    # the path for welding a floor straight weld with v chisels on both sides.
    # start at the right side and move left.
    def calculate_straight_points_floor(struct1, floorthick, leftpointteach, rightpointteach):
        # get the stuff
        point0 = struct1[0]
        p0x = point0[0]
        p0y = point0[1]
        p0z = point0[2]
        v3xunit = struct1[1]
        v3yunit = struct1[2]
        v3zunit = struct1[3]
        heading1 = struct1[4]
        v4xunit = struct1[5]
        v4yunit = struct1[6]
        lpy = leftpointteach[1]
        rpy = rightpointteach[1]

        # first, check if we need a lift column raise
        # (we do not, because the floors are low)
        zpi = p0z
        floorz = zpi

        # calculate pointtopvcham (left point) (tilted and tiltraised)
        chamferup = floorthick * 25.4 / 1000.0
        tiltraise = 0.006 # 6 mm raise needed for the tip to clear the plane during tiltback
        # on this one, move the tiltraise distance sideways (towards robot) and the chamferover distance up
        x = p0x + v4xunit * tiltraise * -1
        y = p0y + v4yunit * tiltraise * -1
        z = floorz + chamferup

        # calculate rxryrz for tilted back
        # 3 rotations to make this happen.
        # start point is straight up with the preheat pointed in the +y direction.
        # first rotation is 90 degrees about y axis. positive direction. gun is now pointing in the x+ direction with preheat facing +y direction
        m1 = get_rotation_matrix_from_description("y", 1, 90 * pi / 180)
        # second rotation is about 180 degrees about the z axis. heading1 plus 90 degrees. gun is now pointing directly into the sidewall
        m2 = get_rotation_matrix_from_description("z", 1, pi/2 + heading1)
        # third rotation is 10 degrees about the z axis. gun is now tilted back 10 degrees from the sidewall
        m3 = get_rotation_matrix_from_description("z", 1, 10 * pi / 180)
        # combine them by multiplying m3 * m2 * m1
        # matrix multiplication is not commutative but it IS associative, so you can do this whichever order
        m4 = multiply_matrix(m2, m1)
        m5 = multiply_matrix(m3, m4)
        rxryrzt = convert_matrix_to_axang(m5)
        rxt = rxryrzt[0]
        ryt = rxryrzt[1]
        rzt = rxryrzt[2]
        # the non tilted angle is just m4
        rxryrz = convert_matrix_to_axang(m4)
        rx = rxryrz[0]
        ry = rxryrz[1]
        rz = rxryrz[2]
        pointtopvcham = p[x, y, z, rxt, ryt, rzt]

        # calculate distance between leftpoint and rightpoint
        # we have the y distance. we need to find the total distance.
        # the unit vector (v3) should have a magnitude of 1. that's what analyze_touchpoints_only_cover_straight() calculated.
        # so the total distance is y distance * 1 / v3yunit
        ydist = rpy - lpy
        totdist = ydist / v3yunit

        # calculate pointtopvcham2 (right point) (tilted and tiltraised)
        x2 = x + v3xunit * totdist
        y2 = y + v3yunit * totdist
        z2 = z + v3zunit * totdist
        pointtopvcham2 = p[x2, y2, z2, rxt, ryt, rzt]

        # calculate point1 (preheat)
        dist = 1 * 25.4 / 1000.0 # move back 1 inch from ptvc2 (in this case back means positive)
        p1x = x2 + dist * v3xunit
        p1y = y2 + dist * v3yunit
        p1z = z2 + dist * v3zunit
        point1 = p[p1x, p1y, p1z, rxt, ryt, rzt]

        # calculate point2 (start of flatten)
        dist = -0.5 * 25.4 / 1000.0  # half an inch past the top of v chamfer
        p2x = x2 + dist * v3xunit
        p2y = y2 + dist * v3yunit
        p2z = z2 + dist * v3zunit
        point2 = p[p2x, p2y, p2z, rxt, ryt, rzt]

        # calculate point3 (end of flatten)
        dist = -1.5 * 25.4 / 1000.0  # 1.5 inches past top of v chamfer
        p3x = x2 + dist * v3xunit + tiltraise * v4xunit
        p3y = y2 + dist * v3yunit + tiltraise * v4yunit
        p3z = z2 + dist * v3zunit
        point3 = p[p3x, p3y, p3z, rx, ry, rz]

        # calculate point4 (start of unflatten)
        dist = 1.5 * 25.4 / 1000.0
        p4x = x + v3xunit * dist + tiltraise * v4xunit
        p4y = y + v3yunit * dist + tiltraise * v4yunit
        p4z = z + v3zunit * dist
        point4 = p[p4x, p4y, p4z, rx, ry, rz]

        # calculate point5 (end of unflatten)
        dist = 0.5 * 25.4 / 1000.0
        p5x = x + v3xunit * dist
        p5y = y + v3yunit * dist
        p5z = z + v3zunit * dist
        point5 = p[p5x, p5y, p5z, rxt, ryt, rzt]

        # calculate point6 (end of smear)
        dist = -2 * 25.4 / 1000.0
        p6x = x + v3xunit * dist
        p6y = y + v3yunit * dist
        p6z = z + v3zunit * dist
        point6 = p[p6x, p6y, p6z, rxt, ryt, rzt]

        # return struct
        ret = struct(pointtopvcham=pointtopvcham, point1=point1, point2=point2, point3=point3, point4=point4, point5=point5, point6=point6)
        return ret

    end

    # this function determines the starting touchpoints for homing in on cover lt geometry
    # includes two points above the cover lt, closer to the robot than the lt, facing down
    def get_coverlt_homing_pathpoints(leftpoint, rightpoint):
        # get the teach position points
        lpx = leftpoint[0]
        lpy = leftpoint[1]
        lpz = leftpoint[2]
        rpx = rightpoint[0]
        rpy = rightpoint[1]
        rpz = rightpoint[2]

        # specify the distances from (in meters)
        d0 = 0.05 # how far from the cover to approach from
        d1 = 0.03 # how far the touchpints are pushed closer to the robot
        d2 = 0.00 # how far inwards the touchpoints are pushed

        # rxryrz
        rxryrz = [0.334, 3.124, 0]
        rx = rxryrz[0]
        ry = rxryrz[1]
        rz = rxryrz[2]

        # calculate the points
        ph1 = p[lpx + d1, lpy + d2, lpz + d0, rx, ry, rz] # left side approach
        ph2 = p[rpx + d1, rpy - d2, rpz + d0, rx, ry, rz] # right side approach

        ret = struct(ph1=ph1, ph2=ph2)
        is_robot_at_reachable_spot(leftpoint, ret)
        return ret
    end

    def main_calculate_cover_lt(p11, p12, leftpoint, rightpoint):
        struct1 = analyze_touchpoints_only_cover_lt(p11, p12, leftpoint, rightpoint)
        struct2 = calculate_points_cover_lt(struct1)
        #struct2 = calculate_DOtA_points_left_extended(struct1, list1, chamferover, chamferup, tcp_pose_top)
        #struct3 = check_validity_left(struct1, struct2)
        return struct2

    end

    def analyze_touchpoints_only_cover_lt(p11, p12, leftpoint, rightpoint):
        # calculate the slope of the groove in xy plane
        l1p1x = leftpoint[0]
        l1p1y = leftpoint[1]
        l1p2x = rightpoint[0]
        l1p2y = rightpoint[1]

        # equate the first line in 2d space
        ml1 = (l1p2y-l1p1y) / (l1p2x-l1p1x)

        # b = y - mx
        bl1 = l1p1y - ml1 * l1p1x

        # zraise (how much the z value changes from left point to right point
        zraise = p12[2] - p11[2]

        #get the calcpoints
        leftcalcpoint = [leftpoint[0], leftpoint[1], p11[2]]
        rightcalcpoint = [rightpoint[0], rightpoint[1], p12[2]]
        # get the vector from a to b
        vec = [rightcalcpoint[0] - leftcalcpoint[0], rightcalcpoint[1] - leftcalcpoint[1], rightcalcpoint[2] - leftcalcpoint[2]]
        # get the unit vector in 3d
        mag3d = sqrt(vec[0]*vec[0]+vec[1]*vec[1]+vec[2]*vec[2])
        vec3dunit = [vec[0]/mag3d, vec[1]/mag3d, vec[2]/mag3d]
        # get the unit vector in 2d
        mag2d = sqrt(vec[0]*vec[0]+vec[1]*vec[1])
        vec2dunit = [vec[0]/mag2d, vec[1]/mag2d]
        # get the heading
        heading1 = convert_uv_to_heading(vec2dunit[0], vec2dunit[1])

        ret = struct(leftcalcpoint=leftcalcpoint, rightcalcpoint=rightcalcpoint, vxunit=vec3dunit[0], vyunit=vec3dunit[1], vzunit=vec3dunit[2], heading1=heading1)
        return ret
    end

    def calculate_points_cover_lt(struct1):
        # get the stuff from struct
        leftcalcpoint = struct1[0]
        x = leftcalcpoint[0]
        y = leftcalcpoint[1]
        z = leftcalcpoint[2]
        rightcalcpoint = struct1[1]
        x2 = rightcalcpoint[0]
        y2 = rightcalcpoint[1]
        z2 = rightcalcpoint[2]
        v3xunit = struct1[2]
        v3yunit = struct1[3]
        v3zunit = struct1[4]
        heading1 = struct1[5]

        # first calculate rxryrz f normal and tiltback
        # calculate rxryrz for tilted back
        # 3 rotations to make this happen.
        # start point is straight up with the preheat pointed in the +y direction.
        # first rotation is 180 degrees about x direction. gun is now pointing straight down with preheat facing -y direction
        m1 = get_rotation_matrix_from_description("x", 1, 180 * pi / 180)
        # second rotation is a 10 degree turn about the x axis (negative direction)
        m2 = get_rotation_matrix_from_description("x", -1, 10 * pi / 180)
        # third rotation is about 180 degrees about the z axis. starting from the -y axis, go until you get to heading1. that will equal heading1 plus 90 degrees
        m3 = get_rotation_matrix_from_description("z", 1, pi/2 + heading1)
        # combine them by multiplying m3 * m2 * m1
        # matrix multiplication is not commutative but it IS associative, so you can do this whichever order
        m4 = multiply_matrix(m2, m1)
        m5 = multiply_matrix(m3, m4)
        rxryrzt = convert_matrix_to_axang(m5)
        rxt = rxryrzt[0]
        ryt = rxryrzt[1]
        rzt = rxryrzt[2]

        # calculate rxryrz for nontilted
        # first rotation is 180 degrees about x direction. gun is now pointing straight down with preheat facing -y direction
        m1 = get_rotation_matrix_from_description("x", 1, 180 * pi / 180)
        # third rotation is about 180 degrees about the z axis. starting from the -y axis, go until you get to heading1. that will equal heading1 plus 90 degrees
        m3 = get_rotation_matrix_from_description("z", 1, pi/2 + heading1)
        m5 = multiply_matrix(m3, m1)
        rxryrz = convert_matrix_to_axang(m5)
        rx = rxryrz[0]
        ry = rxryrz[1]
        rz = rxryrz[2]

        tiltraise = 0.006 # 6 mm raise needed for the tip to clear the plane during tiltback

        # calculate points 1-3
        # calculate point1 (preheat)
        dist = -1 * 25.4 / 1000.0 # move back 1 inch from
        p1x = x + dist * v3xunit
        p1y = y + dist * v3yunit
        p1z = z + dist * v3zunit + tiltraise
        point1 = p[p1x, p1y, p1z, rxt, ryt, rzt]

        # calculate point2 (start of flatten)
        dist = 0.5 * 25.4 / 1000.0  # half an inch past the top of v chamfer
        p2x = x + dist * v3xunit
        p2y = y + dist * v3yunit
        p2z = z + dist * v3zunit + tiltraise
        point2 = p[p2x, p2y, p2z, rxt, ryt, rzt]

        # calculate point3 (end of flatten)
        dist = 1.5 * 25.4 / 1000.0  # 1.5 inches past top of v chamfer
        p3x = x + dist * v3xunit
        p3y = y + dist * v3yunit
        p3z = z + dist * v3zunit
        point3 = p[p3x, p3y, p3z, rx, ry, rz]

        # calculate points 4-6
        # calculate point4 (start of unflatten)
        dist = -1.5 * 25.4 / 1000.0
        p4x = x2 + v3xunit * dist
        p4y = y2 + v3yunit * dist
        p4z = z2 + v3zunit * dist
        point4 = p[p4x, p4y, p4z, rx, ry, rz]

        # calculate point5 (end of unflatten)
        dist = -0.5 * 25.4 / 1000.0
        p5x = x2 + v3xunit * dist
        p5y = y2 + v3yunit * dist
        p5z = z2 + v3zunit * dist + tiltraise
        point5 = p[p5x, p5y, p5z, rxt, ryt, rzt]

        # calculate point6 (end of smear)
        dist = 2 * 25.4 / 1000.0
        p6x = x2 + v3xunit * dist
        p6y = y2 + v3yunit * dist
        p6z = z2 + v3zunit * dist + tiltraise
        point6 = p[p6x, p6y, p6z, rxt, ryt, rzt]

        # return struct
        ret = struct(pointtopvcham=leftcalcpoint, point1=point1, point2=point2, point3=point3, point4=point4, point5=point5, point6=point6)
        return ret

    end

    def main_calculate_sleeve_fillet(p1, p2, p3):
        struct1 = analyze_touchpoints_only_sleeve_fillet(p1, p2, p3)
        struct2 = calculate_points_sleeve_fillet(struct1)
        return struct2
    end

    # given 3 points at the intersection of the sleeve and the sidewall, this calculates and returns 3 things:
    # the centerpoint of the circle on the plane, the normal vector of the plane, and the radius of the circle
    # then it returns 4 more things after converting to a vertical circle/plane: heading1 (into the plane), vecn, vecr, vecu
    def analyze_touchpoints_only_sleeve_fillet(p1, p2, p3):
        x1 = p1[0]
        y1 = p1[1]
        z1 = p1[2]
        x2 = p2[0]
        y2 = p2[1]
        z2 = p2[2]
        x3 = p3[0]
        y3 = p3[1]
        z3 = p3[2]

        # calculate plane
        # calculate ab (1->2) vector
        abvec = [x2-x1, y2-y1, z2-z1]
        # calculate ac (1->3) vector
        acvec = [x3-x1, y3-y1, z3-z1]
        #calculate the plane's normal vector = ab x ac

        n = crossproduct(abvec, acvec)
        mag = sqrt(n[0]*n[0]+n[1]*n[1]+n[2]*n[2])
        n = [n[0]/mag, n[1]/mag, n[2]/mag]
        d = n[0] * x1 + n[1] * y1 + n[2] * z1

        # find the circle
        # Midpoint of AB:
        mab = [(x1 + x2)/2, (y1 + y2)/2, (z1 + z2)/2]
        # midpoint of ac
        mac = [(x3 + x1)/2, (y3 + y1)/2, (z3 + z1)/2]
        # Get Normal Vectors to AB and AC in the Plane
        # nab (normal to ab) = abvec x n
        nab = crossproduct(abvec, n)
        # nac (normal to ac) = acvec x n
        nac = crossproduct(acvec, n)
        # Define Perpendicular Bisector Lines
        # Each line goes through a midpoint and extends in the direction of the na_
        # we already have the equations of those lines in point vector form with l1 = mab + s * nab, and l2 = mac + t * nac
        # define all the terms so the math is simpler when i have to do math
        mabx = mab[0]
        maby = mab[1]
        mabz = mab[2]
        nabx = nab[0]
        naby = nab[1]
        nabz = nab[2]
        macx = mac[0]
        macy = mac[1]
        macz = mac[2]
        nacx = nac[0]
        nacy = nac[1]
        nacz = nac[2]
        # find the intersection point using the y and z equations
        # maby + s * naby = macy + t * nacy
        # mabz + s * nabz = macz + t * nacz
        # first solve for s and take
        # t = (macz*naby + maby*nabz - mabz*naby - macy*nabz) / (nacy*nabz - naby*nacz)
        t = (macz*naby + maby*nabz - mabz*naby - macy*nabz) / (nacy*nabz - naby*nacz)
        # s = (t*nacz + macz - mabz) / nabz
        s = (t*nacz + macz - mabz) / nabz
        # find the point
        # pcenter = mac + t * nac
        pcenterx = macx + t * nacx
        pcentery = macy + t * nacy
        pcenterz = macz + t * nacz
        rxryrz = [0.528, 4.631, 0.258] # demo point of the welder pointing forward into a sleeve
        pcenter = p[pcenterx, pcentery, pcenterz, rxryrz[0], rxryrz[1], rxryrz[2]]
        radius = distance_between(pcenterx, pcentery, pcenterz, x1, y1, z1)

        # ------ start calculation of vertical assumption -----
        # assume the plane close to vertical
        # fix it to make it actually vertical
        # calculate the unit vector of up, and the unit vector of right.
        # calculate the heading from the +x axis to pointing straight into the wall.
        # the unit vector of up is [0, 0, 1] (because the plane is verticalized) (for easier calculations)
        # first calculate the normal vector INTO the sidewall (make sure x is negative) and make it a unit vector
        vecn = [n[0], n[1], 0] # vector normal
        if vecn[0] > 0:
            vecn = [-n[0], -n[1], 0]
        end
        mag = sqrt(vecn[0]*vecn[0]+vecn[1]*vecn[1])
        vecn = [vecn[0]/mag, vecn[1]/mag, 0]
        # next calculate the right normal vector (the vector IN the plane that goes to the right)
        vecr = [vecn[1], -1*vecn[0], 0]
        vecu = [0, 0, 1] # vector up
        heading1 = convert_uv_to_heading(vecn[0], vecn[1])


        ret = struct(pcenter=pcenter, planenormalvec=n, radius=radius, heading1=heading1, vecn=vecn, vecr=vecr, vecu=vecu)
        return ret
    end

    def crossproduct(vec1, vec2):
        nx = vec1[1]*vec2[2] - vec1[2]*vec2[1]
        ny = vec1[2]*vec2[0] - vec1[0]*vec2[2]
        nz = vec1[0]*vec2[1] - vec1[1]*vec2[0]
        ret = [nx, ny, nz]
        return ret
    end

    # this function calculates only the four points of the quadrants, for the not real program.
    # these calculations are easier so that's why i'm starting with them first.
    # this assumes a vertical plane
    def calculate_points_sleeve_fillet_quadonly(struct1):
        # get the stuff from the struct
        pcenter = struct1[0]
        pcx = pcenter[0]
        pcy = pcenter[1]
        pcz = pcenter[2]
        planenormalvec = struct1[1]
        radius = struct1[2]
        heading1 = struct1[3]
        vecn = struct1[4]
        vecnx = vecn[0]
        vecny = vecn[1]
        vecr = struct1[5]
        vecrx = vecr[0]
        vecry = vecr[1]
        vecu = struct1[6]
        vecuz = vecu[2]

        # define cushions (the backofhole can't actually touch the intersection of pipe and wall, it travels a certain distance around it
        cushout = 0.006 # 5mm # the cushion out from the wall
        cusharound = 0.006 # 5mm # the cushion around the sleeve.

        # get the top point (point1)
        # take the center point and move up the radius plus the cushions
        p1x = pcx + vecnx * -1 * cushout
        p1y = pcy + vecny * -1 * cushout
        p1z = pcz + vecuz * radius + vecuz * cusharound

        # find rxryrz1
        # first rotation is 135 degrees about the y- direction. 90 degrees to get flat. Tip pointing x-, preheat pointing y+. 45 more degrees to get at that above angle
        m1 = get_rotation_matrix_from_description("y", -1, 135 * pi / 180)
        # second rotation is heading1 – 180 degrees about the z+ axis to get pointing straight into wall. Heading1 should be about 180 degrees
        m2 = get_rotation_matrix_from_description("z", 1, heading1 - 180 * pi/180)
        # combine them by multiplying
        m3 = multiply_matrix(m2, m1)
        rxryrz1 = convert_matrix_to_axang(m3)
        rx1 = rxryrz1[0]
        ry1 = rxryrz1[1]
        rz1 = rxryrz1[2]

        point1 = p[p1x, p1y, p1z, rx1, ry1, rz1]

        # get second point (right) (point2)
        # take the center point and move right the radius plus the cushions
        p2x = pcx + vecrx * radius + vecrx * cusharound + vecnx * -1 * cushout
        p2y = pcy + vecry * radius + vecry * cusharound + vecny * -1 * cushout
        p2z = pcz

        # find rxryrz2
        # first rotation is 90 degrees about the x- axis
        m1 = get_rotation_matrix_from_description("x", -1, 90 * pi / 180)
        # second rotation is About 135 degrees about the z+ axis. This calculation is heading1 – 45 degrees
        m2 = get_rotation_matrix_from_description("z", 1, heading1 - 45 * pi/180)
        # combine them by multiplying
        m3 = multiply_matrix(m2, m1)
        rxryrz2 = convert_matrix_to_axang(m3)
        rx2 = rxryrz2[0]
        ry2 = rxryrz2[1]
        rz2 = rxryrz2[2]

        point2 = p[p2x, p2y, p2z, rx2, ry2, rz2]

        # get the third point (bottom) (point3)
        p3x = pcx + vecnx * -1 * cushout
        p3y = pcy + vecny * -1 * cushout
        p3z = pcz - vecuz * radius - vecuz * cusharound

        # find rxryrz3
        # first rotation is 45 degrees about the y+ axis
        m1 = get_rotation_matrix_from_description("y", 1, 45 * pi / 180)
        # second rotation is About 180 degrees about the z+ axis. This calculation is heading1 degrees
        m2 = get_rotation_matrix_from_description("z", 1, heading1)
        # combine them by multiplying
        m3 = multiply_matrix(m2, m1)
        rxryrz3 = convert_matrix_to_axang(m3)
        rx3 = rxryrz3[0]
        ry3 = rxryrz3[1]
        rz3 = rxryrz3[2]

        point3 = p[p3x, p3y, p3z, rx3, ry3, rz3]

        # get the fourth point (left) (point4)
        p4x = pcx - vecrx * radius - vecrx * cusharound + vecnx * -1 * cushout
        p4y = pcy - vecry * radius - vecry * cusharound + vecny * -1 * cushout
        p4z = pcz

        # find rxryrz4
        # first rotation is 90 degrees about the x+ axis
        m1 = get_rotation_matrix_from_description("x", 1, 90 * pi / 180)
        # second rotation is heading1 + 45 degrees about the z+ axis. approx 225 degrees ccw
        m2 = get_rotation_matrix_from_description("z", 1, heading1 + 45 * pi/180)
        # combine them by multiplying
        m3 = multiply_matrix(m2, m1)
        rxryrz4 = convert_matrix_to_axang(m3)
        rx4 = rxryrz4[0]
        ry4 = rxryrz4[1]
        rz4 = rxryrz4[2]

        point4 = p[p4x, p4y, p4z, rx4, ry4, rz4]

        # return the points
        ret = struct(point1=point1, point2=point2, point3=point3, point4=point4)
        return ret

    end

    # this function calculates the points necessary for the fillet sleeve weld path.
    # this assumes a vertical plane
    def calculate_points_sleeve_fillet(struct1):
        # get the stuff from the struct
        pcenter = struct1[0]
        pcx = pcenter[0]
        pcy = pcenter[1]
        pcz = pcenter[2]
        planenormalvec = struct1[1]
        radius = struct1[2]
        heading1 = struct1[3]
        vecn = struct1[4]
        vecnx = vecn[0]
        vecny = vecn[1]
        vecr = struct1[5]
        vecrx = vecr[0]
        vecry = vecr[1]
        vecu = struct1[6]
        vecuz = vecu[2]

        # define cushions (the backofhole can't actually touch the intersection of pipe and wall, it travels a certain distance around it
        cushout = 0.006 # 5mm # the cushion out from the wall
        cusharound = 0.006 # 5mm # the cushion around the sleeve.

        # get the top point (point1)
        # take the center point and move up the radius plus the cushions
        p1x = pcx + vecnx * -1 * cushout
        p1y = pcy + vecny * -1 * cushout
        p1z = pcz + vecuz * radius + vecuz * cusharound

        # find rxryrz1
        # first rotation is 135 degrees about the y- direction. 90 degrees to get flat. Tip pointing x-, preheat pointing y+. 45 more degrees to get at that above angle
        m1 = get_rotation_matrix_from_description("y", -1, 135 * pi / 180)
        # second rotation is heading1 – 180 degrees about the z+ axis to get pointing straight into wall. Heading1 should be about 180 degrees
        m2 = get_rotation_matrix_from_description("z", 1, heading1 - 180 * pi/180)
        # combine them by multiplying
        m3 = multiply_matrix(m2, m1)
        rxryrz1 = convert_matrix_to_axang(m3)
        rx1 = rxryrz1[0]
        ry1 = rxryrz1[1]
        rz1 = rxryrz1[2]

        point1 = p[p1x, p1y, p1z, rx1, ry1, rz1]

        # get second point (right) (point2)
        # take the center point and move right the radius plus the cushions
        p2x = pcx + vecrx * radius + vecrx * cusharound + vecnx * -1 * cushout
        p2y = pcy + vecry * radius + vecry * cusharound + vecny * -1 * cushout
        p2z = pcz

        # find rxryrz2
        # first rotation is 90 degrees about the x- axis
        m1 = get_rotation_matrix_from_description("x", -1, 90 * pi / 180)
        # second rotation is About 135 degrees about the z+ axis. This calculation is heading1 – 45 degrees
        m2 = get_rotation_matrix_from_description("z", 1, heading1 - 45 * pi/180)
        # combine them by multiplying
        m3 = multiply_matrix(m2, m1)
        rxryrz2 = convert_matrix_to_axang(m3)
        rx2 = rxryrz2[0]
        ry2 = rxryrz2[1]
        rz2 = rxryrz2[2]

        point2 = p[p2x, p2y, p2z, rx2, ry2, rz2]

        # get the third point (bottom) (point3)
        p3x = pcx + vecnx * -1 * cushout
        p3y = pcy + vecny * -1 * cushout
        p3z = pcz - vecuz * radius - vecuz * cusharound

        # find rxryrz3
        # first rotation is 45 degrees about the y+ axis
        m1 = get_rotation_matrix_from_description("y", 1, 45 * pi / 180)
        # second rotation is About 180 degrees about the z+ axis. This calculation is heading1 degrees
        m2 = get_rotation_matrix_from_description("z", 1, heading1)
        # combine them by multiplying
        m3 = multiply_matrix(m2, m1)
        rxryrz3 = convert_matrix_to_axang(m3)
        rx3 = rxryrz3[0]
        ry3 = rxryrz3[1]
        rz3 = rxryrz3[2]

        point3 = p[p3x, p3y, p3z, rx3, ry3, rz3]

        # get the fourth point (left) (point4)
        p4x = pcx - vecrx * radius - vecrx * cusharound + vecnx * -1 * cushout
        p4y = pcy - vecry * radius - vecry * cusharound + vecny * -1 * cushout
        p4z = pcz

        # find rxryrz4
        # first rotation is 90 degrees about the x+ axis
        m1 = get_rotation_matrix_from_description("x", 1, 90 * pi / 180)
        # second rotation is heading1 + 45 degrees about the z+ axis. approx 225 degrees ccw
        m2 = get_rotation_matrix_from_description("z", 1, heading1 + 45 * pi/180)
        # combine them by multiplying
        m3 = multiply_matrix(m2, m1)
        rxryrz4 = convert_matrix_to_axang(m3)
        rx4 = rxryrz4[0]
        ry4 = rxryrz4[1]
        rz4 = rxryrz4[2]

        point4 = p[p4x, p4y, p4z, rx4, ry4, rz4]

        # get the angle for the tilt-back at the top (p1)
        m0 = get_rotation_matrix_from_description("x", -1, 10 * pi / 180)
        m1 = get_rotation_matrix_from_description("y", -1, 135 * pi / 180)
        # second rotation is heading1 – 180 degrees about the z+ axis to get pointing straight into wall. Heading1 should be about 180 degrees
        m2 = get_rotation_matrix_from_description("z", 1, heading1 - 180 * pi/180)
        # combine them by multiplying
        m3 = multiply_matrix(m2, m1)
        m4 = multiply_matrix(m3, m0)
        rxryrz1tilt = convert_matrix_to_axang(m4)
        rx1t = rxryrz1tilt[0]
        ry1t = rxryrz1tilt[1]
        rz1t = rxryrz1tilt[2]

        # point 1, but with the tilt back angle
        point1t = p[p1x, p1y, p1z, rx1t, ry1t, rz1t]

        # point45 (the point 45 degrees along the path) (has no rxryrz data) (because if we do fixed angle circle move it wont use that anyways, it'l just use the angle from p1t)
        distup = cos(45 * pi/180) * (radius + cusharound)
        distover = sin(45 * pi/180) * (radius + cusharound)
        p45x = pcx + vecrx * distover + vecnx * -1 * cushout
        p45y = pcy + vecry * distover + vecny * -1 * cushout
        p45z = pcz + vecuz * distup
        point45 = p[p45x, p45y, p45z, 0,0,0]

        # point22 (22.5 degrees of angle)
        distup = cos(22.5 * pi/180) * (radius + cusharound)
        distover = sin(22.5 * pi/180) * (radius + cusharound)
        p22x = pcx + vecrx * distover + vecnx * -1 * cushout
        p22y = pcy + vecry * distover + vecny * -1 * cushout
        p22z = pcz + vecuz * distup
        point22 = p[p22x, p22y, p22z, 0,0,0]

        # return the points
        ret = struct(point1=point1, point2=point2, point3=point3, point4=point4, point1t=point1t, point45=point45, point22=point22)
        return ret

    end
    $ 391 "'list possible points'"
    # 'list possible points'
    $ 392 "robot 1 moves"
    $ 393 "If 1≟2"
    if (1 == 2):
      $ 394 "MoveJ"
      $ 395 "r1_ek_oldhome" "breakAfter"
      movej(get_inverse_kin(r1_ek_oldhome_p, qnear=r1_ek_oldhome_q), a=1.3962634015954636, v=1.0471975511965976)
      $ 396 "r1_ek_extrude" "breakAfter"
      movej(get_inverse_kin(r1_ek_extrude_p, qnear=r1_ek_extrude_q), a=1.3962634015954636, v=1.0471975511965976)
      $ 397 "r1_ek_front" "breakAfter"
      movej(get_inverse_kin(r1_ek_front_p, qnear=r1_ek_front_q), a=1.3962634015954636, v=1.0471975511965976)
      $ 398 "r1_ek_middle" "breakAfter"
      movej(get_inverse_kin(r1_ek_middle_p, qnear=r1_ek_middle_q), a=1.3962634015954636, v=1.0471975511965976)
      $ 399 "r1_ek_middle2" "breakAfter"
      movej(get_inverse_kin(r1_ek_middle2_p, qnear=r1_ek_middle2_q), a=1.3962634015954636, v=1.0471975511965976)
      $ 400 "r1_ek_bottom" "breakAfter"
      movej(get_inverse_kin(r1_ek_bottom_p, qnear=r1_ek_bottom_q), a=1.3962634015954636, v=1.0471975511965976)
      $ 401 "r1_ek_end" "breakAfter"
      movej(get_inverse_kin(r1_ek_end_p, qnear=r1_ek_end_q), a=1.3962634015954636, v=1.0471975511965976)
    end
    $ 402 "robot 2 moves"
    $ 403 "If 1≟2"
    if (1 == 2):
      $ 404 "MoveJ"
      $ 405 "r2_ek_oldhome" "breakAfter"
      movej(get_inverse_kin(r2_ek_oldhome_p, qnear=r2_ek_oldhome_q), a=1.3962634015954636, v=1.0471975511965976)
      $ 407 "r2_ek_extrude" "breakAfter"
      movej(get_inverse_kin(r2_ek_extrude_p, qnear=r2_ek_extrude_q), a=1.3962634015954636, v=1.0471975511965976)
      $ 408 "r2_ek_front" "breakAfter"
      movej(get_inverse_kin(r2_ek_front_p, qnear=r2_ek_front_q), a=1.3962634015954636, v=1.0471975511965976)
      $ 409 "r2_ek_middle" "breakAfter"
      movej(get_inverse_kin(r2_ek_middle_p, qnear=r2_ek_middle_q), a=1.3962634015954636, v=1.0471975511965976)
      $ 410 "r2_ek_bottom" "breakAfter"
      movej(get_inverse_kin(r2_ek_bottom_p, qnear=r2_ek_bottom_q), a=1.3962634015954636, v=1.0471975511965976)
      $ 411 "r2_ek_end" "breakAfter"
      movej(get_inverse_kin(r2_ek_end_p, qnear=r2_ek_end_q), a=1.3962634015954636, v=1.0471975511965976)
    end
    $ 412 "'detemine correct points for which robot'"
    # 'detemine correct points for which robot'
    $ 413 "If robot_number≟1"
    if (robot_number == 1):
      $ 414 "robot1 positions"
      $ 415 "ek_oldhome≔r1_ek_oldhome_p"
      global ek_oldhome=r1_ek_oldhome_p
      $ 416 "ek_extrude≔r1_ek_extrude_p"
      global ek_extrude=r1_ek_extrude_p
      $ 417 "ek_front≔r1_ek_front_p"
      global ek_front=r1_ek_front_p
      $ 418 "ek_middle≔r1_ek_middle_p"
      global ek_middle=r1_ek_middle_p
      $ 419 "ek_middle2≔r1_ek_middle2_p"
      global ek_middle2=r1_ek_middle2_p
      $ 420 "ek_bottom≔r1_ek_bottom_p"
      global ek_bottom=r1_ek_bottom_p
      $ 421 "ek_end≔r1_ek_end_q"
      global ek_end=r1_ek_end_q
    else:
      $ 422 "ElseIf robot_number≟2"
      if (robot_number == 2):
        $ 423 "robot1 positions"
        $ 424 "ek_oldhome≔r2_ek_oldhome_p"
        global ek_oldhome=r2_ek_oldhome_p
        $ 425 "ek_extrude≔r2_ek_extrude_p"
        global ek_extrude=r2_ek_extrude_p
        $ 426 "ek_front≔r2_ek_front_p"
        global ek_front=r2_ek_front_p
        $ 427 "ek_middle≔r2_ek_middle_p"
        global ek_middle=r2_ek_middle_p
        $ 428 "ek_middle2≔r2_ek_middle_p"
        global ek_middle2=r2_ek_middle_p
        $ 429 "ek_bottom≔r2_ek_bottom_p"
        global ek_bottom=r2_ek_bottom_p
        $ 430 "ek_end≔r2_ek_end_q"
        global ek_end=r2_ek_end_q
      end
    end
    $ 431 "'start of program'"
    # 'start of program'
    $ 433 "Set"
    set_tcp(p[-0.00588,-0.33377999999999997,0.10496,1.2092,-1.2092,1.2092])
    $ 434 "MoveJ"
    $ 436 "ek_oldhome" "breakAfter"
    movej(ek_oldhome, a=1.3962634015954636, v=1.0471975511965976)
    $ 437 "'above waypoint is home'"
    # 'above waypoint is home'
    $ 438 "'move above bucket'"
    # 'move above bucket'
    $ 439 "MoveJ"
    $ 441 "ek_extrude" "breakAfter"
    movej(ek_extrude, a=1.3962634015954636, v=1.0471975511965976)
    $ 442 "'extrude out a foot'"
    # 'extrude out a foot'
    # begin: URCap Program Node
    #   Source: WireTank Serial, 4.9.0, WireTank, LLC
    #   Type: WireTank Serial
    $ 444 "Serial Bridge uR1"
    SerialResponse = WTSerialBridge.send_command("/dev/ttyUSB0",1200, 8, "None", "One", "None", 1000, "None", "None", [252,82,49], False)
    # end: URCap Program Node
    $ 445 "Set DO[0]=On"
    set_standard_digital_out(0, True)
    $ 446 "Wait: 24.0"
    sleep(24.0)
    # begin: URCap Program Node
    #   Source: WireTank Serial, 4.9.0, WireTank, LLC
    #   Type: WireTank Serial
    $ 447 "Serial Bridge uR0"
    SerialResponse = WTSerialBridge.send_command("/dev/ttyUSB0",1200, 8, "None", "One", "None", 1000, "None", "None", [252,82,48], False)
    # end: URCap Program Node
    $ 448 "Wait: 1.0"
    sleep(1.0)
    $ 449 "Set DO[0]=Off"
    set_standard_digital_out(0, False)
    $ 450 "'slice'"
    # 'slice'
    $ 451 "MoveL"
    $ 457 "ek_front" "breakAfter"
    movel(ek_front, a=0.05, v=0.03)
    $ 458 "ek_middle" "breakAfter"
    movel(ek_middle, a=0.05, v=0.03)
    $ 459 "ek_middle2" "breakAfter"
    movel(ek_middle2, a=0.05, v=0.03)
    $ 460 "ek_bottom" "breakAfter"
    movel(ek_bottom, a=0.05, v=0.03)
    $ 461 "ek_end" "breakAfter"
    movel(ek_end, a=0.05, v=0.03)
    $ 462 "MoveJ"
    $ 464 "ek_oldhome" "breakAfter"
    movej(ek_oldhome, a=1.3962634015954636, v=1.0471975511965976)
    $ 465 "'above waypoint is home'"
    # 'above waypoint is home'
  end
  def align_tcp_forward():
    $ 467 "align_tcp_forward" "noBreak"
    $ 468 "'this program aligns the tcp parallel to the y direction'"
    # 'this program aligns the tcp parallel to the y direction'
    $ 469 "cp≔get_actual_tcp_pose()"
    global cp= get_actual_tcp_pose ()
    $ 470 "aligned_y_pose≔p[cp[0],cp[1],cp[2],0,-1.570796,0]"
    global aligned_y_pose=p[cp[0],cp[1],cp[2],0,-1.570796,0]
    $ 471 "MoveJ"
    $ 472 "aligned_y_pose" "breakAfter"
    movej(aligned_y_pose, a=1.3962634015954636, v=1.0471975511965976)
  end
  def align_tcp_up():
    $ 473 "align_tcp_up" "noBreak"
    $ 474 "'this program aligns the tcp parallel to the y direction'"
    # 'this program aligns the tcp parallel to the y direction'
    $ 475 "cp≔get_actual_tcp_pose()"
    global cp= get_actual_tcp_pose ()
    $ 476 "aligned_y_pose≔p[cp[0],cp[1],cp[2],0,0,0]"
    global aligned_y_pose=p[cp[0],cp[1],cp[2],0,0,0]
    $ 477 "MoveJ"
    $ 478 "aligned_y_pose" "breakAfter"
    movej(aligned_y_pose, a=1.3962634015954636, v=1.0471975511965976)
  end
  def align_ready_for_welding():
    $ 479 "align_ready_for_welding" "noBreak"
    $ 480 "'this program takes the welder from home to a position alined ready for welding (vertically down)'"
    # 'this program takes the welder from home to a position alined ready for welding (vertically down)'
    $ 481 "MoveJ"
    $ 482 "oldhome" "breakAfter"
    movej(get_inverse_kin(oldhome_p, qnear=oldhome_q), a=1.3962634015954636, v=1.0471975511965976)
    $ 483 "Waypoint_34" "breakAfter"
    movej(get_inverse_kin(Waypoint_34_p, qnear=Waypoint_34_q), a=1.3962634015954636, v=1.0471975511965976)
    $ 484 "Waypoint_35" "breakAfter"
    movej(get_inverse_kin(Waypoint_35_p, qnear=Waypoint_35_q), a=1.3962634015954636, v=1.0471975511965976)
    $ 485 "Waypoint_36" "breakAfter"
    movej(get_inverse_kin(Waypoint_36_p, qnear=Waypoint_36_q), a=1.3962634015954636, v=1.0471975511965976)
  end
  def Corner_Homing_45():
    $ 486 "Corner_Homing_45" "noBreak"
    $ 487 "'Use this program when tool is already positioned close to corner at 45deg'"
    # 'Use this program when tool is already positioned close to corner at 45deg'
    $ 488 "'tool flange will seek all 3 sides. will save those 5 locs in p__'"
    # 'tool flange will seek all 3 sides. will save those 5 locs in p__'
    $ 489 "Set"
    set_tcp(p[1.4000000000000001E-4,-0.01751,0.284,0.0,0.0,0.0])
    $ 498 "Wait: 1.0"
    sleep(1.0)
    $ 499 "tp≔get_actual_tcp_pose()"
    global tp= get_actual_tcp_pose ()
    $ 503 "path_pre≔get_corner_homing_45_pathpoints(tp,tcp_pose_top)"
    global path_pre=get_corner_homing_45_pathpoints(tp,tcp_pose_top)
    $ 504 "ph1≔path_pre[0]"
    global ph1=path_pre[0]
    $ 505 "ph2≔path_pre[1]"
    global ph2=path_pre[1]
    $ 506 "ph3≔path_pre[2]"
    global ph3=path_pre[2]
    $ 507 "ph4≔path_pre[3]"
    global ph4=path_pre[3]
    $ 508 "ph5≔path_pre[4]"
    global ph5=path_pre[4]
    $ 509 "ph6≔path_pre[5]"
    global ph6=path_pre[5]
    $ 510 "ph7≔path_pre[6]"
    global ph7=path_pre[6]
    $ 511 "ph2up≔path_pre[7]"
    global ph2up=path_pre[7]
    $ 512 "ph4up≔path_pre[8]"
    global ph4up=path_pre[8]
    $ 513 "MoveL"
    $ 514 "ph1" "breakAfter"
    movel(ph1, a=0.2, v=0.25)
    $ 515 "ph2" "breakAfter"
    movel(ph2, a=0.2, v=0.25)
    $ 516 "MoveL"
    $ 517 "Direction: Base"
    global move_thread_flag_517=0
    thread move_thread_517():
      enter_critical
      move_thread_flag_517 = 1
      local towardsPos=calculate_point_to_move_towards(p[0.0,0.0,0.0,0.0,0.0,0.0], [-1,-1.0,0.0], 1000.0)
      movel(towardsPos, a=0.1, v=0.02)
      move_thread_flag_517 = 2
      exit_critical
    end
    move_thread_flag_517 = 0
    move_thread_han_517 = run move_thread_517()
    while (True):
      local targetTcpDirection=get_target_tcp_speed()
      local stepsToRetract=tool_contact(direction=targetTcpDirection)
      if (stepsToRetract > 0):
        kill move_thread_han_517
        stopl(3.0)
        local backTrackMovement=get_actual_joint_positions_history(stepsToRetract)
        local contactPose=get_forward_kin(backTrackMovement)
        local posDir=[targetTcpDirection[0],targetTcpDirection[1],targetTcpDirection[2]]
        local retractTo=contactPose
        if (norm(posDir) > 1e-6):
          local normalizedPosDir=normalize(posDir)
          local additionalRetraction=p[normalizedPosDir[0] * 0.0, normalizedPosDir[1] * 0.0, normalizedPosDir[2] * 0.0, 0, 0, 0]
          retractTo = pose_sub(contactPose, additionalRetraction)
        end
        movel(retractTo, a=3.0, v=0.1)
        $ 518 "Until (tool_contact_detection)"
        break
      end
      sync()
    end
    $ 519 "p11≔get_actual_tcp_pose()"
    global p11= get_actual_tcp_pose ()
    $ 520 "MoveJ"
    $ 521 "ph2" "breakAfter"
    movej(ph2, a=1.3962634015954636, v=1.0471975511965976)
    $ 522 "ph2up" "breakAfter"
    movej(ph2up, a=1.3962634015954636, v=1.0471975511965976)
    $ 523 "MoveL"
    $ 524 "Direction: Base"
    global move_thread_flag_524=0
    thread move_thread_524():
      enter_critical
      move_thread_flag_524 = 1
      local towardsPos=calculate_point_to_move_towards(p[0.0,0.0,0.0,0.0,0.0,0.0], [-1,-1.0,0.0], 1000.0)
      movel(towardsPos, a=0.1, v=0.02)
      move_thread_flag_524 = 2
      exit_critical
    end
    move_thread_flag_524 = 0
    move_thread_han_524 = run move_thread_524()
    while (True):
      local targetTcpDirection=get_target_tcp_speed()
      local stepsToRetract=tool_contact(direction=targetTcpDirection)
      if (stepsToRetract > 0):
        kill move_thread_han_524
        stopl(3.0)
        local backTrackMovement=get_actual_joint_positions_history(stepsToRetract)
        local contactPose=get_forward_kin(backTrackMovement)
        local posDir=[targetTcpDirection[0],targetTcpDirection[1],targetTcpDirection[2]]
        local retractTo=contactPose
        if (norm(posDir) > 1e-6):
          local normalizedPosDir=normalize(posDir)
          local additionalRetraction=p[normalizedPosDir[0] * 0.0, normalizedPosDir[1] * 0.0, normalizedPosDir[2] * 0.0, 0, 0, 0]
          retractTo = pose_sub(contactPose, additionalRetraction)
        end
        movel(retractTo, a=3.0, v=0.1)
        $ 525 "Until (tool_contact_detection)"
        break
      end
      sync()
    end
    $ 526 "p13≔get_actual_tcp_pose()"
    global p13= get_actual_tcp_pose ()
    $ 527 "MoveJ"
    $ 528 "ph2up" "breakAfter"
    movej(ph2up, a=1.3962634015954636, v=1.0471975511965976)
    $ 529 "ph3" "breakAfter"
    movej(ph3, a=1.3962634015954636, v=1.0471975511965976)
    $ 530 "MoveL"
    $ 531 "Direction: Base"
    global move_thread_flag_531=0
    thread move_thread_531():
      enter_critical
      move_thread_flag_531 = 1
      local towardsPos=calculate_point_to_move_towards(p[0.0,0.0,0.0,0.0,0.0,0.0], [-1,-1.0,0.0], 1000.0)
      movel(towardsPos, a=0.1, v=0.02)
      move_thread_flag_531 = 2
      exit_critical
    end
    move_thread_flag_531 = 0
    move_thread_han_531 = run move_thread_531()
    while (True):
      local targetTcpDirection=get_target_tcp_speed()
      local stepsToRetract=tool_contact(direction=targetTcpDirection)
      if (stepsToRetract > 0):
        kill move_thread_han_531
        stopl(3.0)
        local backTrackMovement=get_actual_joint_positions_history(stepsToRetract)
        local contactPose=get_forward_kin(backTrackMovement)
        local posDir=[targetTcpDirection[0],targetTcpDirection[1],targetTcpDirection[2]]
        local retractTo=contactPose
        if (norm(posDir) > 1e-6):
          local normalizedPosDir=normalize(posDir)
          local additionalRetraction=p[normalizedPosDir[0] * 0.0, normalizedPosDir[1] * 0.0, normalizedPosDir[2] * 0.0, 0, 0, 0]
          retractTo = pose_sub(contactPose, additionalRetraction)
        end
        movel(retractTo, a=3.0, v=0.1)
        $ 532 "Until (tool_contact_detection)"
        break
      end
      sync()
    end
    $ 533 "p12≔get_actual_tcp_pose()"
    global p12= get_actual_tcp_pose ()
    $ 537 "MoveJ"
    $ 538 "ph3" "breakAfter"
    movej(ph3, a=1.3962634015954636, v=1.0471975511965976)
    $ 539 "ph1" "breakAfter"
    movej(ph1, a=1.3962634015954636, v=1.0471975511965976)
    $ 544 "MoveL"
    $ 545 "ph4" "breakAfter"
    movel(ph4, a=1.2, v=0.25)
    $ 546 "MoveL"
    $ 547 "Direction: Base"
    global move_thread_flag_547=0
    thread move_thread_547():
      enter_critical
      move_thread_flag_547 = 1
      local towardsPos=calculate_point_to_move_towards(p[0.0,0.0,0.0,0.0,0.0,0.0], [-1.0,1.0,0.0], 1000.0)
      movel(towardsPos, a=0.1, v=0.02)
      move_thread_flag_547 = 2
      exit_critical
    end
    move_thread_flag_547 = 0
    move_thread_han_547 = run move_thread_547()
    while (True):
      local targetTcpDirection=get_target_tcp_speed()
      local stepsToRetract=tool_contact(direction=targetTcpDirection)
      if (stepsToRetract > 0):
        kill move_thread_han_547
        stopl(3.0)
        local backTrackMovement=get_actual_joint_positions_history(stepsToRetract)
        local contactPose=get_forward_kin(backTrackMovement)
        local posDir=[targetTcpDirection[0],targetTcpDirection[1],targetTcpDirection[2]]
        local retractTo=contactPose
        if (norm(posDir) > 1e-6):
          local normalizedPosDir=normalize(posDir)
          local additionalRetraction=p[normalizedPosDir[0] * 0.0, normalizedPosDir[1] * 0.0, normalizedPosDir[2] * 0.0, 0, 0, 0]
          retractTo = pose_sub(contactPose, additionalRetraction)
        end
        movel(retractTo, a=3.0, v=0.1)
        $ 548 "Until (tool_contact_detection)"
        break
      end
      sync()
    end
    $ 549 "p21≔get_actual_tcp_pose()"
    global p21= get_actual_tcp_pose ()
    $ 550 "MoveL"
    $ 551 "ph4" "breakAfter"
    movel(ph4, a=1.2, v=0.25)
    $ 552 "ph4up" "breakAfter"
    movel(ph4up, a=1.2, v=0.25)
    $ 553 "MoveL"
    $ 554 "Direction: Base"
    global move_thread_flag_554=0
    thread move_thread_554():
      enter_critical
      move_thread_flag_554 = 1
      local towardsPos=calculate_point_to_move_towards(p[0.0,0.0,0.0,0.0,0.0,0.0], [-1.0,1.0,0.0], 1000.0)
      movel(towardsPos, a=0.1, v=0.02)
      move_thread_flag_554 = 2
      exit_critical
    end
    move_thread_flag_554 = 0
    move_thread_han_554 = run move_thread_554()
    while (True):
      local targetTcpDirection=get_target_tcp_speed()
      local stepsToRetract=tool_contact(direction=targetTcpDirection)
      if (stepsToRetract > 0):
        kill move_thread_han_554
        stopl(3.0)
        local backTrackMovement=get_actual_joint_positions_history(stepsToRetract)
        local contactPose=get_forward_kin(backTrackMovement)
        local posDir=[targetTcpDirection[0],targetTcpDirection[1],targetTcpDirection[2]]
        local retractTo=contactPose
        if (norm(posDir) > 1e-6):
          local normalizedPosDir=normalize(posDir)
          local additionalRetraction=p[normalizedPosDir[0] * 0.0, normalizedPosDir[1] * 0.0, normalizedPosDir[2] * 0.0, 0, 0, 0]
          retractTo = pose_sub(contactPose, additionalRetraction)
        end
        movel(retractTo, a=3.0, v=0.1)
        $ 555 "Until (tool_contact_detection)"
        break
      end
      sync()
    end
    $ 556 "p23≔get_actual_tcp_pose()"
    global p23= get_actual_tcp_pose ()
    $ 557 "MoveL"
    $ 558 "ph4up" "breakAfter"
    movel(ph4up, a=1.2, v=0.25)
    $ 559 "ph5" "breakAfter"
    movel(ph5, a=1.2, v=0.25)
    $ 560 "MoveL"
    $ 561 "Direction: Base"
    global move_thread_flag_561=0
    thread move_thread_561():
      enter_critical
      move_thread_flag_561 = 1
      local towardsPos=calculate_point_to_move_towards(p[0.0,0.0,0.0,0.0,0.0,0.0], [-1.0,1.0,0.0], 1000.0)
      movel(towardsPos, a=0.1, v=0.02)
      move_thread_flag_561 = 2
      exit_critical
    end
    move_thread_flag_561 = 0
    move_thread_han_561 = run move_thread_561()
    while (True):
      local targetTcpDirection=get_target_tcp_speed()
      local stepsToRetract=tool_contact(direction=targetTcpDirection)
      if (stepsToRetract > 0):
        kill move_thread_han_561
        stopl(3.0)
        local backTrackMovement=get_actual_joint_positions_history(stepsToRetract)
        local contactPose=get_forward_kin(backTrackMovement)
        local posDir=[targetTcpDirection[0],targetTcpDirection[1],targetTcpDirection[2]]
        local retractTo=contactPose
        if (norm(posDir) > 1e-6):
          local normalizedPosDir=normalize(posDir)
          local additionalRetraction=p[normalizedPosDir[0] * 0.0, normalizedPosDir[1] * 0.0, normalizedPosDir[2] * 0.0, 0, 0, 0]
          retractTo = pose_sub(contactPose, additionalRetraction)
        end
        movel(retractTo, a=3.0, v=0.1)
        $ 562 "Until (tool_contact_detection)"
        break
      end
      sync()
    end
    $ 563 "p22≔get_actual_tcp_pose()"
    global p22= get_actual_tcp_pose ()
    $ 574 "MoveJ"
    $ 575 "ph5" "breakAfter"
    movej(ph5, a=1.3962634015954636, v=1.0471975511965976)
    $ 576 "MoveL"
    $ 577 "ph4" "breakAfter"
    movel(ph4, a=1.2, v=0.25)
    $ 578 "ph1" "breakAfter"
    movel(ph1, a=1.2, v=0.25)
    $ 579 "MoveJ"
    $ 580 "Waypoint_4" "breakAfter"
    movej(get_inverse_kin(Waypoint_4_p, qnear=Waypoint_4_q), a=1.3962634015954636, v=1.0471975511965976)
    $ 581 "Waypoint_13" "breakAfter"
    movej(get_inverse_kin(Waypoint_13_p, qnear=Waypoint_13_q), a=1.3962634015954636, v=1.0471975511965976)
    $ 582 "Waypoint_1" "breakAfter"
    movej(get_inverse_kin(Waypoint_1_p, qnear=Waypoint_1_q), a=1.3962634015954636, v=1.0471975511965976)
    $ 583 "ph6" "breakAfter"
    movej(ph6, a=1.3962634015954636, v=1.0471975511965976)
    $ 584 "ph7" "breakAfter"
    movej(ph7, a=1.3962634015954636, v=1.0471975511965976)
    $ 585 "Wait: 1.0"
    sleep(1.0)
    $ 589 "MoveL"
    $ 590 "Direction: Base Z+"
    global move_thread_flag_590=0
    thread move_thread_590():
      enter_critical
      move_thread_flag_590 = 1
      local towardsPos=calculate_point_to_move_towards(p[0.0,0.0,0.0,0.0,0.0,0.0], [0.0,0.0,1.0], 1000.0)
      movel(towardsPos, a=0.1, v=0.02)
      move_thread_flag_590 = 2
      exit_critical
    end
    move_thread_flag_590 = 0
    move_thread_han_590 = run move_thread_590()
    while (True):
      local targetTcpDirection=get_target_tcp_speed()
      local stepsToRetract=tool_contact(direction=targetTcpDirection)
      if (stepsToRetract > 0):
        kill move_thread_han_590
        stopl(3.0)
        local backTrackMovement=get_actual_joint_positions_history(stepsToRetract)
        local contactPose=get_forward_kin(backTrackMovement)
        local posDir=[targetTcpDirection[0],targetTcpDirection[1],targetTcpDirection[2]]
        local retractTo=contactPose
        if (norm(posDir) > 1e-6):
          local normalizedPosDir=normalize(posDir)
          local additionalRetraction=p[normalizedPosDir[0] * 0.0, normalizedPosDir[1] * 0.0, normalizedPosDir[2] * 0.0, 0, 0, 0]
          retractTo = pose_sub(contactPose, additionalRetraction)
        end
        movel(retractTo, a=3.0, v=0.1)
        $ 591 "Until (tool_contact_detection)"
        break
      end
      sync()
    end
    $ 592 "p3≔get_actual_tcp_pose()"
    global p3= get_actual_tcp_pose ()
    $ 593 "MoveJ"
    $ 594 "ph7" "breakAfter"
    movej(ph7, a=1.3962634015954636, v=1.0471975511965976)
    $ 595 "ph6" "breakAfter"
    movej(ph6, a=1.3962634015954636, v=1.0471975511965976)
    $ 596 "Waypoint_14" "breakAfter"
    movej(get_inverse_kin(Waypoint_14_p, qnear=Waypoint_14_q), a=1.3962634015954636, v=1.0471975511965976)
    $ 597 "Waypoint_4" "breakAfter"
    movej(get_inverse_kin(Waypoint_4_p, qnear=Waypoint_4_q), a=1.3962634015954636, v=1.0471975511965976)
    $ 598 "Waypoint_41" "breakAfter"
    movej(get_inverse_kin(Waypoint_41_p, qnear=Waypoint_41_q), a=1.3962634015954636, v=1.0471975511965976)
    $ 599 "'above waypoint is home'"
    # 'above waypoint is home'
    $ 601 "Comment"
    # Comment
    $ 602 "Comment"
    # Comment
    $ 603 "Comment"
    # Comment
    $ 604 "Comment"
    # Comment
    $ 605 "Comment"
    # Comment
    $ 606 "Comment"
    # Comment
  end
  $ 2 "BeforeStart"
  $ 3 "Safe Home Folder"
  $ 4 "'if robot is not at home, send it back to home safely'"
  # 'if robot is not at home, send it back to home safely'
  $ 5 "'make sure the tcp is welder'"
  # 'make sure the tcp is welder'
  $ 6 "Set"
  set_tcp(p[-0.0095,-0.328,0.105,1.2092,-1.2092,1.2092])
  $ 7 "sp≔get_actual_tcp_pose()"
  global sp= get_actual_tcp_pose ()
  $ 8 "MoveL"
  $ 9 "sp" "breakAfter"
  movel(sp, a=1.2, v=0.25)
  $ 10 "'if first move is to a variable, skip automove'"
  # 'if first move is to a variable, skip automove'
  $ 11 "'turn off welder'"
  # 'turn off welder'
  # begin: URCap Program Node
  #   Source: WireTank Serial, 4.9.0, WireTank, LLC
  #   Type: WireTank Serial
  $ 12 "Serial Bridge uR0"
  SerialResponse = WTSerialBridge.send_command("/dev/ttyUSB0",1200, 8, "None", "One", "None", 1000, "None", "None", [252,82,48], False)
  # end: URCap Program Node
  $ 13 "Set DO[0]=Off"
  set_standard_digital_out(0, False)
  $ 14 "jp≔get_actual_joint_positions()"
  global jp= get_actual_joint_positions ()
  $ 15 "If sp[0]>0.600"
  if (sp[0]>0.600):
    $ 16 "'if x > 600 then above then home'"
    # 'if x > 600 then above then home'
    $ 17 "MoveJ"
    $ 19 "Waypoint_76" "breakAfter"
    movej(get_inverse_kin(Waypoint_76_p, qnear=Waypoint_76_q), a=1.3962634015954636, v=1.0471975511965976)
    $ 20 "Home"
    movej([-3.266929759358355, -1.2139462677784536, 1.5878387874396154, 1.1069165929565088, -0.0023738326664366483, -1.7891447305770605], a=1.3962634015954636, v=1.0471975511965976)
  else:
    $ 21 "Else" "noBreak"
    $ 22 "Popup: retreating to home"
    popup("retreating to home", "Message", False, False, blocking=True)
    $ 23 "'for rules 2-8, finish with oldhome then above then home'"
    # 'for rules 2-8, finish with oldhome then above then home'
    $ 24 "If -1.74<jp[4] and jp[4]<1.05 and -1.74<jp[3] and jp[3]<1.74"
    if (-1.74<jp[4]  and  jp[4]<1.05  and  -1.74<jp[3]  and  jp[3]<1.74):
      $ 25 "'if oldhome, test teach, then go straight to oldhome'"
      # 'if oldhome, test teach, then go straight to oldhome'
    else:
      $ 26 "ElseIf sp[0]<-.5 and jp[3]>3.14 and -2.62<jp[4] and jp[4]<-0.87"
      if (sp[0]<-.5  and  jp[3]>3.14  and  -2.62<jp[4]  and  jp[4]<-0.87):
        $ 27 "'if left side weld approach, left weld approach in reverse'"
        # 'if left side weld approach, left weld approach in reverse'
        $ 28 "MoveJ"
        $ 29 "Waypoint_50" "breakAfter"
        movej(get_inverse_kin(Waypoint_50_p, qnear=Waypoint_50_q), a=1.3962634015954636, v=1.0471975511965976)
        $ 30 "Waypoint_51" "breakAfter"
        movej(get_inverse_kin(Waypoint_51_p, qnear=Waypoint_51_q), a=1.3962634015954636, v=1.0471975511965976)
        $ 31 "Waypoint_52" "breakAfter"
        movej(get_inverse_kin(Waypoint_52_p, qnear=Waypoint_52_q), a=1.3962634015954636, v=1.0471975511965976)
        $ 32 "Waypoint_53" "breakAfter"
        movej(get_inverse_kin(Waypoint_53_p, qnear=Waypoint_53_q), a=1.3962634015954636, v=1.0471975511965976)
      else:
        $ 33 "ElseIf sp[0]<0 and 0<jp[3] and jp[3]<1.74 and 0.87<jp[4] and jp[4]<2.62"
        if (sp[0]<0  and  0<jp[3]  and  jp[3]<1.74  and  0.87<jp[4]  and  jp[4]<2.62):
          $ 34 "'if right side around, move back then wapoint 24 then oldhome'"
          # 'if right side around, move back then wapoint 24 then oldhome'
          $ 35 "If sp[0]<-1.0"
          if (sp[0]<-1.0):
            $ 36 "xback≔p[-1.0,sp[1],sp[2],sp[3],sp[4],sp[5]]"
            global xback=p[-1.0,sp[1],sp[2],sp[3],sp[4],sp[5]]
            $ 37 "MoveJ"
            $ 38 "xback" "breakAfter"
            movej(xback, a=1.3962634015954636, v=1.0471975511965976)
          end
          $ 39 "MoveJ"
          $ 40 "Waypoint_54" "breakAfter"
          movej(get_inverse_kin(Waypoint_54_p, qnear=Waypoint_54_q), a=1.3962634015954636, v=1.0471975511965976)
        else:
          $ 41 "ElseIf jp[3]>2.62 and jp[4]<-3.84"
          if (jp[3]>2.62  and  jp[4]<-3.84):
            $ 42 "'if left side second half, then left weld ending sequence'"
            # 'if left side second half, then left weld ending sequence'
            $ 43 "If jp[5]<0.35"
            if (jp[5]<0.35):
              $ 44 "MoveJ"
              $ 45 "Waypoint_65" "breakAfter"
              movej(get_inverse_kin(Waypoint_65_p, qnear=Waypoint_65_q), a=1.3962634015954636, v=1.0471975511965976)
            end
            $ 46 "MoveJ"
            $ 51 "'above is testing, below is real'"
            # 'above is testing, below is real'
            $ 52 "Waypoint_55" "breakAfter"
            movej(get_inverse_kin(Waypoint_55_p, qnear=Waypoint_55_q), a=1.3962634015954636, v=1.0471975511965976)
            $ 54 "Waypoint_59" "breakAfter"
            movej(get_inverse_kin(Waypoint_59_p, qnear=Waypoint_59_q), t=2.0)
            $ 55 "Waypoint_71" "breakAfter"
            movej(get_inverse_kin(Waypoint_71_p, qnear=Waypoint_71_q), a=1.3962634015954636, v=1.0471975511965976)
            $ 56 "Waypoint_58" "breakAfter"
            movej(get_inverse_kin(Waypoint_58_p, qnear=Waypoint_58_q), a=1.3962634015954636, v=1.0471975511965976)
            $ 57 "Waypoint_56" "breakAfter"
            movej(get_inverse_kin(Waypoint_56_p, qnear=Waypoint_56_q), a=1.3962634015954636, v=1.0471975511965976)
            $ 58 "Waypoint_57" "breakAfter"
            movej(get_inverse_kin(Waypoint_57_p, qnear=Waypoint_57_q), a=1.3962634015954636, v=1.0471975511965976)
          else:
            $ 59 "ElseIf jp[3]<-2.09"
            if (jp[3]<-2.09):
              $ 60 "'bottom homing'"
              # 'bottom homing'
              $ 61 "MoveJ"
              $ 63 "Comment"
              # Comment
              $ 64 "If sp[0]<-0.95"
              if (sp[0]<-0.95):
                $ 65 "xback≔p[-0.95,sp[1],sp[2],sp[3],sp[4],sp[5]]"
                global xback=p[-0.95,sp[1],sp[2],sp[3],sp[4],sp[5]]
                $ 66 "MoveL"
                $ 67 "xback" "breakAfter"
                movel(xback, a=1.2, v=0.25)
              end
              $ 68 "Waypoint_67" "breakAfter"
              movej(get_inverse_kin(Waypoint_67_p, qnear=Waypoint_67_q), a=1.3962634015954636, v=1.0471975511965976)
            else:
              $ 69 "ElseIf jp[3]<0 and jp[4]<-3.14"
              if (jp[3]<0  and  jp[4]<-3.14):
                $ 70 "'if left side homing, special unspin'"
                # 'if left side homing, special unspin'
                $ 71 "MoveJ"
                $ 73 "Comment"
                # Comment
                $ 74 "Waypoint_69" "breakAfter"
                movej(get_inverse_kin(Waypoint_69_p, qnear=Waypoint_69_q), a=1.3962634015954636, v=1.0471975511965976)
                $ 75 "Waypoint_70" "breakAfter"
                movej(get_inverse_kin(Waypoint_70_p, qnear=Waypoint_70_q), a=1.3962634015954636, v=1.0471975511965976)
              else:
                $ 76 "ElseIf (sp[4]<-3 or sp[4]>3) and -0.02<sp[5] and sp[5]<0.02"
                if ((sp[4]<-3  or  sp[4]>3)  and  -0.02<sp[5]  and  sp[5]<0.02):
                  $ 77 "'go straight to home'"
                  # 'go straight to home'
                else:
                  $ 78 "ElseIf 2>1"
                  if (2>1):
                    $ 79 "'if none of the other options, then error continuously'"
                    # 'if none of the other options, then error continuously'
                    $ 80 "Loop 2>1"
                    while (2>1):
                      $ 81 "Popup: Unknown Position. Find Calvin for Assistance"
                      popup("Unknown Position. Find Calvin for Assistance", "Message", False, False, blocking=True)
                    end
                  end
                end
              end
            end
          end
        end
      end
    end
    $ 82 "'insert logic for how to get back to oldhome'"
    # 'insert logic for how to get back to oldhome'
    $ 83 "'finish with oldhome then above then home'"
    # 'finish with oldhome then above then home'
    $ 84 "MoveJ"
    $ 85 "Waypoint_49" "breakAfter"
    movej(get_inverse_kin(Waypoint_49_p, qnear=Waypoint_49_q), a=1.3962634015954636, v=1.0471975511965976)
    $ 87 "Waypoint_75" "breakAfter"
    movej(get_inverse_kin(Waypoint_75_p, qnear=Waypoint_75_q), a=1.3962634015954636, v=1.0471975511965976)
    $ 88 "Home"
    movej([-3.266929759358355, -1.2139462677784536, 1.5878387874396154, 1.1069165929565088, -0.0023738326664366483, -1.7891447305770605], a=1.3962634015954636, v=1.0471975511965976)
    # begin: URCap Program Node
    #   Source: MachineLogic for Universal Robots, 3.1.7, Vention Inc.
    #   Type: MachineLogic for Universal Robots
    $ 89 "MachineLogic Homing"
    while isVentionMovementBusyMachineMotion1==True:
    sleep(0.05)
    end
    if(isVentionMovementBusyMachineMotion1 == False):
    isVentionMovementBusyMachineMotion1 = True
    socket_send_string("estop/status;", "MachineMotion1")
    temp_estop_var_vention = socket_read_string("MachineMotion1",timeout=15)
    while(temp_estop_var_vention=="estop/status true"):
    if temp_estop_var_vention=="estop/status true":
    sendStringWithTimeout("estop/systemreset/request","Ack estop/systemreset/request;","MachineMotion1")
    end
    socket_send_string("estop/status;", "MachineMotion1")
    temp_estop_var_vention = socket_read_string("MachineMotion1",timeout=15)
    if temp_estop_var_vention=="estop/status true":
    popup("MachineMotion in estop, make sure you have all emergency modules released manually. If you continue the system will try to reset MachineMotion automatically.",blocking=True)
    end
    end
    else:
    popup("resource is being used already: MachineMotion1")
    halt
    end
    isVentionMovementBusyMachineMotion1 = True
    sendString("im_home_axis_1", "MachineMotion im_home_axis_1 = completed", "MachineMotion1")
    isVentionMovementBusyMachineMotion1 = False
    sendString("SET im_set_encoder_pos_aux_1 0.000", "Ack", "MachineMotion1")
    isVentionMovementBusyMachineMotion1 = False
    sleep(0.03)
    # end: URCap Program Node
  end
  $ 607 "Thread_1"
  thread Thread_1():
    $ 608 "Loop  True "
    while (  True  ):
      $ 609 "If freedrive_m_var≟ True "
      if (freedrive_m_var ==   True  ):
        $ 610 "freedrive_mode()"
        freedrive_mode()
        $ 611 "free_dr_already≔ True "
        global free_dr_already=  True
      else:
        $ 612 "Else" "noBreak"
        $ 613 "If free_dr_already"
        if (free_dr_already):
          $ 614 "end_freedrive_mode()"
          end_freedrive_mode()
        end
      end
      $ 615 "sync()"
      sync()
    end
  end
  threadId_Thread_1 = run Thread_1()
  $ 90 "Robot Program"
  $ 91 "'start of main program'"
  # 'start of main program'
  $ 92 "Set"
  set_tcp(p[-0.0095,-0.328,0.105,1.2092,-1.2092,1.2092])
  $ 93 "Home"
  movej([-3.266929759358355, -1.2139462677784536, 1.5878387874396154, 1.1069165929565088, -0.0023738326664366483, -1.7891447305770605], a=1.3962634015954636, v=1.0471975511965976)
  $ 94 "Script: analyze_touchpoints.script"
  # this file creates the function for analyzing touchpoints
  # define pi
  pi = 3.1415926535
  # initialize a lift column extension needed of 0.0
  global liftcolumnzneeded = 0.0

  # this is the main entry point for calculations.
  # it takes in the 5 points, analyzes the shape of the box, and then calculates path points and returns them
  # specifically for Down, Over, then Around (DOtA)
  # specifically for right-sided boxes (vertical weld on right side of edge)
  def main_calculate_right(p11, p12, p21, p22, p3, p13, p23, chamferover):
      struct1 = analyze_touchpoints_only(p11, p12, p21, p22, p3)
      list1 = analyze_vertical_touchpoints(p11, p12, p13, p21, p22, p23, p3)
      struct2 = calculate_DOtA_points_right(struct1, list1, chamferover)
      validity = check_validity_right(struct1, struct2)
      return struct2
  end

  # this is the main entry point for calculations.
  # it takes in the 5 points, analyzes the shape of the box, and then calculates path points and returns them
  # specifically for Down, Over, then Around (DOtA)
  # specifically for left-sided boxes (vertical weld on left side of edge)
  def main_calculate_left(p11, p12, p21, p22, p3, p13, p23, chamferover):
      struct1 = analyze_touchpoints_only(p11, p12, p21, p22, p3)
      list1 = analyze_vertical_touchpoints(p11, p12, p13, p21, p22, p23, p3)
      struct2 = calculate_DOtA_points_left(struct1, list1, chamferover)
      validity = check_validity_left(struct1, struct2)
      return struct2
  end

  # this is the main entry point for calculations, for Floor Corner Extended.
  # it takes in the 7 touchpoints, analyzes the shape of the box.
  # takes in the user defined point for the top of the weld (tcp_pose_top) and then calculates path points
  # loopingly tries to calculate the extension along the sidewall that fulfills get_inverse_kin_has_solution() and provides the farthest extension possible
  # returns the pathpoints
  # specifically for Down, Over, then Around (DOtA)
  # specifically for right-sided boxes (vertical weld on right side of edge)
  def main_calculate_right_extended(p11, p12, p21, p22, p3, p13, p23, chamferover, chamferup, tcp_pose_top):
      struct1 = analyze_touchpoints_only(p11, p12, p21, p22, p3)
      list1 = analyze_vertical_touchpoints(p11, p12, p13, p21, p22, p23, p3)
      struct2 = calculate_DOtA_points_right_extended(struct1, list1, chamferover, chamferup, tcp_pose_top)
      struct3 = check_validity_right(struct1, struct2)
      return struct3
  end

  # this is the main entry point for calculations, for Floor Corner Extended.
  # it takes in the 7 touchpoints, analyzes the shape of the box.
  # takes in the user defined point for the top of the weld (tcp_pose_top) and then calculates path points
  # loopingly tries to calculate the extension along the sidewall that fulfills get_inverse_kin_has_solution() and provides the farthest extension possible
  # returns the pathpoints
  # specifically for Down, Over, then Around (DOtA)
  # specifically for left-sided boxes (vertical weld on left side of edge)
  def main_calculate_left_extended(p11, p12, p21, p22, p3, p13, p23, chamferover, chamferup, tcp_pose_top):
      struct1 = analyze_touchpoints_only(p11, p12, p21, p22, p3)
      list1 = analyze_vertical_touchpoints(p11, p12, p13, p21, p22, p23, p3)
      struct2 = calculate_DOtA_points_left_extended(struct1, list1, chamferover, chamferup, tcp_pose_top)
      struct3 = check_validity_left(struct1, struct2)
      return struct3
  end

  # it takes 5 arguments as points
  # it returns a struct containing: (pointintersect, pointapproach1, pointapproach2, point1, point2, point3, point4, point5, pointreturn1, heading1, heading2, heading3, path2r1, path2r2, path2l1, path2l2)
  # specifically for Around then Up (AtU)
  def analyze_touchpoints(p11, p12, p21, p22, p3):
    # FIND THE INTERSECTION
    # comment get the z
    zcoord=p3[2]

    # get the raw points from the first line
    l1p1x=p11[0]
    l1p1y=p11[1]
    l1p2x=p12[0]
    l1p2y=p12[1]

    # equate the first line in 2d space
    ml1 = (l1p2y-l1p1y) / (l1p2x-l1p1x)

    # b = y - mx
    bl1 = l1p1y - ml1 * l1p1x

    # get the raw points from the second line
    l2p1x=p21[0]
    l2p1y=p21[1]
    l2p2x=p22[0]
    l2p2y=p22[1]

    # equate the second line in 2d space
    ml2 = (l2p2y-l2p1y) / (l2p2x-l2p1x)

    # b = y - mx
    bl2 = l2p1y - ml2 * l2p1x


    # find the intersection of the two lines
    # m1x+b1 = m2x+b2
    # m1x - m2x = b2 - b1
    # x = (b2-b1) / (m1-m2)
    xintersect = (bl2-bl1) / (ml1-ml2)
    yintersect = ml1 * xintersect + bl1

    #FIND THE VECTORS
    #define a vector from the intersection to the second point on the first line
    l1delxfull = l1p2x - xintersect
    l1delyfull = l1p2y - yintersect

    l1delmag = sqrt(l1delxfull*l1delxfull + l1delyfull*l1delyfull)

    l1delxunit = l1delxfull / l1delmag
    l1delyunit = l1delyfull / l1delmag

    #define a vector from the intersection to the second point on the second line
    l2delxfull = l2p2x - xintersect
    l2delyfull = l2p2y - yintersect

    l2delmag = sqrt(l2delxfull*l2delxfull + l2delyfull*l2delyfull)

    l2delxunit = l2delxfull / l2delmag
    l2delyunit = l2delyfull / l2delmag

    # FIND THE FOUR POINTS ON THE LINES
    # find locations 8 inches away from  intersect point
    # CONST
    welddistance = 8
    roundoverdistance = 0.05
    zup = .375
    # inches
    wd = welddistance * 25.4 / 1000
    rod = roundoverdistance * 25.4 / 1000
    zup = zup * 25.4 / 1000

    # now we have the unit vector. extend the weld distance from the intersection
    x = xintersect + l1delxunit * wd
    y = yintersect + l1delyunit * wd
    z = zcoord + zup

    point1 = p[x,y,z,1.570796,0,0] # dummy orientation for now

    x = xintersect + l1delxunit * rod
    y = yintersect + l1delyunit * rod

    point2 = p[x,y,z,1.570796,0,0]

    # now we have the unit vector. extend the weld distance from the intersection
    x = xintersect + l2delxunit * wd
    y = yintersect + l2delyunit * wd

    point5 = p[x,y,z,0,-1.570796,0]

    x = xintersect + l2delxunit * rod
    y = yintersect + l2delyunit * rod

    point4 = p[x,y,z,0,-1.570796,0]

    #DEFINE APPROACH POINTS
    pointintersect = p[xintersect,yintersect,zcoord,0,0,0]
    pointapproach1 = p[xintersect+0.1,yintersect+0.1,z,1.570796,0,0]
    pointapproach2 = p[point1[0], point1[1]+0.1, point1[2], point1[3], point1[4], point1[5]]
    pointreturn1 = p[point5[0]+0.1, point5[1], point5[2], point5[3], point5[4], point5[5]]

    #FIND HEADINGS
    #for each heading, find the angle of the line with respect to the pos x axis. then add/subtract 90 degrees because you want to be perpendicular to that
    headingvector1 = convert_uv_to_heading(l1delxunit, l1delyunit)
    headingvector2 = convert_uv_to_heading(l2delxunit, l2delyunit)
    # find halfway heading
    heading2 = (headingvector1 + headingvector2)/2
    # find headings that the robot should face while traveling, perpendicular to the vectors of the sides of the box
    heading1 = headingvector1 + pi/2
    heading3 = headingvector2 - pi/2

    #FIND POINT 3
    #see if we have to / can find point 3
    findpoint3 = True
    if roundoverdistance == 0:
      findpoint3 = False
    end
    if findpoint3:
      # i need to find the point3 such that the arc from p2 to p3 to p4 is tangent to p1-p2 and p4-p5. making this a smooth path will be good
      # the direction of movement is from pointintersect in the direction of heading2
      # how much movement though? this will depend on whether it is actually a 90 degree angle or not.
      # first, find the perpendicular lines through points 2 and 4
      perp2 = find_perpendicular_line(ml1, point2[0], point2[1])
      perp4 = find_perpendicular_line(ml2, point4[0], point4[1])
      # next, find the intersection of those two lines
      perpintersect = find_intersection(perp2[0], perp2[1], perp4[0], perp4[1])
      radiusofcircle = distance_between(perpintersect[0], perpintersect[1], 0, point2[0], point2[1], 0)
      # find a vector the direction of heading2
      uvx = cos(heading2)
      uvy = sin(heading2)
      # compute point3. pass in negative radius because the direction is into the tank but we want to move from the intersection out to the rounded edge
      point3coords = add_vectordistance_to_point(perpintersect[0], perpintersect[1], z, uvx, uvy, 0, -1 * radiusofcircle)
      point3 = p[point3coords[0], point3coords[1], point3coords[2], 0, 0, 0]
    end

    #APPLY ACTUAL RXRYRZ TO POINTS
    # convert the headings to rxryrz and insert those values into the relevant points
    rxryrz = convert_heading_to_axang(heading1)
    rx = rxryrz[0]
    ry = rxryrz[1]
    rz = rxryrz[2]
    pointapproach1 = p[pointapproach1[0], pointapproach1[1], pointapproach1[2], rx, ry, rz]
    pointapproach2 = p[pointapproach2[0], pointapproach2[1], pointapproach2[2], rx, ry, rz]
    point1 = p[point1[0], point1[1], point1[2], rx, ry, rz]
    point2 = p[point2[0], point2[1], point2[2], rx, ry, rz]
    rxryrz = convert_heading_to_axang(heading2)
    rx = rxryrz[0]
    ry = rxryrz[1]
    rz = rxryrz[2]
    if findpoint3:
      point3 = p[point3[0], point3[1], point3[2], rx, ry, rz]
    else:
      point3 = point2
    end
    rxryrz = convert_heading_to_axang(heading3)
    rx = rxryrz[0]
    ry = rxryrz[1]
    rz = rxryrz[2]
    point4 = p[point4[0], point4[1], point4[2], rx, ry, rz]
    point5 = p[point5[0], point5[1], point5[2], rx, ry, rz]
    pointreturn1 = p[pointreturn1[0], pointreturn1[1], pointreturn1[2], rx, ry, rz]

    #find path2 (the part that goes up)
    four_vertical_points = find_vertical_points(pointintersect, l1delxunit, l1delyunit, l2delxunit, l2delyunit, zup, wd, heading1, heading3)
    path2r1 = four_vertical_points[0]
    path2r2 = four_vertical_points[1]
    path2l1 = four_vertical_points[2]
    path2l2 = four_vertical_points[3]

    #RETURN STRUCT
    ret = struct(pointintersect=pointintersect, pointapproach1=pointapproach1, pointapproach2=pointapproach2, point1=point1, point2=point2, point3=point3, point4=point4, point5=point5, pointreturn1=pointreturn1, heading1=heading1, heading2=heading2, heading3=heading3, path2r1=path2r1, path2r2=path2r2, path2l1=path2l1, path2l2=path2l2)
    return ret
  end

  # based on a Corner Homing 45 Cover pattern of touchpoints
  # this uses those touchpoints to create a representation of the corner in 3d robot space.
  def analyze_touchpoints_only_cover(p11, p12, p21, p3):
      zcoord=p3[2]

      # get the raw points from the first line
      l1p1x=p11[0]
      l1p1y=p11[1]
      l1p2x=p12[0]
      l1p2y=p12[1]

      # equate the first line in 2d space
      ml1 = (l1p2y-l1p1y) / (l1p2x-l1p1x)

      # b = y - mx
      bl1 = l1p1y - ml1 * l1p1x

      # get the raw points from the second line
      l2p1x=p21[0]
      l2p1y=p21[1]

      # equate the second line in 2d space
      # ml2 = opposite reciprocal of ml1 (because they are perpendicular) (assume perpendicular to make calculation of weldpath much easier)
      ml2 = -1 / ml1

      # b = y - mx
      bl2 = l2p1y - ml2 * l2p1x

      # find the intersection of the two lines
      # m1x+b1 = m2x+b2
      # m1x - m2x = b2 - b1
      # x = (b2-b1) / (m1-m2)
      xintersect = (bl2-bl1) / (ml1-ml2)
      yintersect = ml1 * xintersect + bl1

      pointintersect = p[xintersect,yintersect,zcoord,0,0,0]

      #FIND THE VECTORS
      #define a vector from the intersection to the second point on the first line
      l1delxfull = l1p2x - xintersect
      l1delyfull = l1p2y - yintersect

      l1delmag = sqrt(l1delxfull*l1delxfull + l1delyfull*l1delyfull)

      l1delxunit = l1delxfull / l1delmag
      l1delyunit = l1delyfull / l1delmag

      #define a vector from the intersection to the second point on the second line
      l2delxfull = l2p1x - xintersect
      l2delyfull = l2p1y - yintersect

      l2delmag = sqrt(l2delxfull*l2delxfull + l2delyfull*l2delyfull)

      l2delxunit = l2delxfull / l2delmag
      l2delyunit = l2delyfull / l2delmag

      #FIND HEADINGS
      #for each heading, find the angle of the line with respect to the pos x axis. this line is from pointintersect and along each edge of the corner
      heading1 = convert_uv_to_heading(l1delxunit, l1delyunit)
      heading3 = convert_uv_to_heading(l2delxunit, l2delyunit)
      # find halfway heading
      heading2 = (heading1 + heading3)/2

      #RETURN STRUCT
      ret = struct(pointintersect=pointintersect, heading1=heading1, heading2=heading2, heading3=heading3, l1delxunit=l1delxunit, l1delyunit=l1delyunit, l2delxunit=l2delxunit, l2delyunit=l2delyunit)
      return ret
  end

  # it takes 5 arguments as points
  # it returns a struct containing: (pointintersect, heading1, heading2, heading3, l1delxunit, l1delyunit, l2delxunit, l2delyunit)
  def analyze_touchpoints_only(p11, p12, p21, p22, p3):
    # FIND THE INTERSECTION
    # comment get the z
    zcoord=p3[2]

    # get the raw points from the first line
    l1p1x=p11[0]
    l1p1y=p11[1]
    l1p2x=p12[0]
    l1p2y=p12[1]

    # equate the first line in 2d space
    ml1 = (l1p2y-l1p1y) / (l1p2x-l1p1x)

    # b = y - mx
    bl1 = l1p1y - ml1 * l1p1x

    # get the raw points from the second line
    l2p1x=p21[0]
    l2p1y=p21[1]
    l2p2x=p22[0]
    l2p2y=p22[1]

    # equate the second line in 2d space
    ml2 = (l2p2y-l2p1y) / (l2p2x-l2p1x)

    # b = y - mx
    bl2 = l2p1y - ml2 * l2p1x


    # find the intersection of the two lines
    # m1x+b1 = m2x+b2
    # m1x - m2x = b2 - b1
    # x = (b2-b1) / (m1-m2)
    xintersect = (bl2-bl1) / (ml1-ml2)
    yintersect = ml1 * xintersect + bl1

    pointintersect = p[xintersect,yintersect,zcoord,0,0,0]

    #FIND THE VECTORS
    #define a vector from the intersection to the second point on the first line
    l1delxfull = l1p2x - xintersect
    l1delyfull = l1p2y - yintersect

    l1delmag = sqrt(l1delxfull*l1delxfull + l1delyfull*l1delyfull)

    l1delxunit = l1delxfull / l1delmag
    l1delyunit = l1delyfull / l1delmag

    #define a vector from the intersection to the second point on the second line
    l2delxfull = l2p2x - xintersect
    l2delyfull = l2p2y - yintersect

    l2delmag = sqrt(l2delxfull*l2delxfull + l2delyfull*l2delyfull)

    l2delxunit = l2delxfull / l2delmag
    l2delyunit = l2delyfull / l2delmag

    #FIND HEADINGS
    #for each heading, find the angle of the line with respect to the pos x axis. then add/subtract 90 degrees because you want to be perpendicular to that
    headingvector1 = convert_uv_to_heading(l1delxunit, l1delyunit)
    headingvector2 = convert_uv_to_heading(l2delxunit, l2delyunit)
    # find halfway heading
    heading2 = (headingvector1 + headingvector2)/2
    # find headings that the robot should face while traveling, perpendicular to the vectors of the sides of the box
    heading1 = headingvector1 + pi/2
    heading3 = headingvector2 - pi/2

    #RETURN STRUCT
    ret = struct(pointintersect=pointintersect, heading1=heading1, heading2=heading2, heading3=heading3, l1delxunit=l1delxunit, l1delyunit=l1delyunit, l2delxunit=l2delxunit, l2delyunit=l2delyunit)
    return ret
  end

  # given a struct from analyze_touchpoints_only(), calculate the points
  # for right, for non-extended
  def calculate_DOtA_points_right(struct1, listleans, chamferover):
      # get the stuff from the struct
      pointintersect = struct1[0]
      heading1 = struct1[1]
      heading2 = struct1[2]
      heading3 = struct1[3]
      l1delxunit = struct1[4]
      l1delyunit = struct1[5]
      l2delxunit = struct1[6]
      l2delyunit = struct1[7]

      # FIND THE POINTS ON THE LINES OF THE FIRST TURN PATH
      # find locations 8 inches away from  intersect point
      # CONST
      welddistance1 = 8 # vertical weld distance
      welddistance2 = 6 # first path second leg
      welddistance3 = 8 # second path second leg
      zup = .375
      # inches
      wd1 = welddistance1 * 25.4 / 1000
      wd2 = welddistance2 * 25.4 / 1000
      wd3 = welddistance3 * 25.4 / 1000
      zup = zup * 25.4 / 1000
      chamferovermm =  chamferover * 25.4 / 1000

      x = pointintersect[0] + l1delxunit * chamferovermm
      y = pointintersect[1] + l1delyunit * chamferovermm
      z = pointintersect[2] + zup

      #apply actual rxryrz to points
      # convert the headings to rxryrz and insert those values into the relevant points
      rxryrz = convert_heading_to_axang_preheatdown(heading1)
      rx = rxryrz[0]
      ry = rxryrz[1]
      rz = rxryrz[2]

      point1 = p[x + wd1*listleans[0], y + wd1*listleans[1], z + wd1, rx, ry, rz] # add in the listleans factor to follow the face of the box as we move up
      point2 = p[x, y, z, rx, ry, rz]

      # convert the headings to rxryrz and insert those values into the relevant points
      rxryrz = convert_heading_to_axang_ccw(heading1)
      rx = rxryrz[0]
      ry = rxryrz[1]
      rz = rxryrz[2]

      point4 = p[x, y, z, rx, ry, rz]
      x = x + l1delxunit * wd2
      y = y + l1delyunit * wd2
      point5 = p[x, y, z, rx, ry, rz]

      # FIND THE POINTS ON THE LINES OF THE SECOND AROUND PATH
      roundoverdistance = 0.05
      rod = roundoverdistance * 25.4 / 1000

      # now we have the unit vector. extend the weld distance from the intersection
      x = pointintersect[0] + l1delxunit * chamferovermm
      y = pointintersect[1] + l1delyunit * chamferovermm
      # convert the headings to rxryrz and insert those values into the relevant points
      rxryrz = convert_heading_to_axang(heading1)
      rx = rxryrz[0]
      ry = rxryrz[1]
      rz = rxryrz[2]
      point_1 = p[x, y, z, rx, ry, rz]

      x = pointintersect[0] + l1delxunit * rod
      y = pointintersect[1] + l1delyunit * rod
      point_2 = p[x, y, z, rx, ry, rz]

      # now we have the unit vector. extend the weld distance from the intersection
      x = pointintersect[0] + l2delxunit * wd3
      y = pointintersect[1] + l2delyunit * wd3
      # convert the headings to rxryrz and insert those values into the relevant points
      rxryrz = convert_heading_to_axang(heading3)
      rx = rxryrz[0]
      ry = rxryrz[1]
      rz = rxryrz[2]
      point_5 = p[x, y, z, rx, ry, rz]

      x = pointintersect[0] + l2delxunit * rod
      y = pointintersect[1] + l2delyunit * rod
      point_4 = p[x, y, z, rx, ry, rz]

      #FIND POINT 3
      # by calling analyze_touchpoints()
      atret = analyze_touchpoints(point_2, point_1, point_4, point_5, pointintersect)
      point_3 = atret[5]


      struct2 = struct(point1=point1, point2=point2, point4=point4, point5=point5, point_1=point_1, point_2=point_2, point_3=point_3, point_4=point_4, point_5=point_5)
      return struct2
  end

  # given a struct from analyze_touchpoints_only(), calculate the points
  # for left, for non-extended
  def calculate_DOtA_points_left(struct1, listleans, chamferover):
      # get the stuff from the struct
      pointintersect = struct1[0]
      heading1 = struct1[1]
      heading2 = struct1[2]
      heading3 = struct1[3]
      l1delxunit = struct1[4]
      l1delyunit = struct1[5]
      l2delxunit = struct1[6]
      l2delyunit = struct1[7]

      # FIND THE POINTS ON THE LINES OF THE FIRST TURN PATH
      # find locations 8 inches away from  intersect point
      # CONST
      welddistance1 = 8 # vertical weld distance
      welddistance2 = 6 # first path second leg
      welddistance3 = 8 # second path second leg
      zup = .375
      # inches
      wd1 = welddistance1 * 25.4 / 1000
      wd2 = welddistance2 * 25.4 / 1000
      wd3 = welddistance3 * 25.4 / 1000
      zup = zup * 25.4 / 1000
      chamferovermm =  chamferover * 25.4 / 1000

      x = pointintersect[0] + l2delxunit * chamferovermm
      y = pointintersect[1] + l2delyunit * chamferovermm
      z = pointintersect[2] + zup

      #apply actual rxryrz to points
      # convert the headings to rxryrz and insert those values into the relevant points
      rxryrz = convert_heading_to_axang_preheatdown(heading3)
      rx = rxryrz[0]
      ry = rxryrz[1]
      rz = rxryrz[2]

      point1 = p[x + wd1*listleans[0], y + wd1*listleans[1], z + wd1, rx, ry, rz]
      point2 = p[x, y, z, rx, ry, rz]

      # convert the headings to rxryrz and insert those values into the relevant points
      rxryrz = convert_heading_to_axang(heading3)
      rx = rxryrz[0]
      ry = rxryrz[1]
      rz = rxryrz[2]

      point4 = p[x, y, z, rx, ry, rz]
      x = x + l2delxunit * wd2
      y = y + l2delyunit * wd2
      point5 = p[x, y, z, rx, ry, rz]

      # FIND THE POINTS ON THE LINES OF THE SECOND AROUND PATH
      roundoverdistance = 0.05
      rod = roundoverdistance * 25.4 / 1000

      # now we have the unit vector. extend the weld distance from the intersection
      x = pointintersect[0] + l2delxunit * chamferovermm
      y = pointintersect[1] + l2delyunit * chamferovermm
      # convert the headings to rxryrz and insert those values into the relevant points
      rxryrz = convert_heading_to_axang_ccw(heading3)
      rx = rxryrz[0]
      ry = rxryrz[1]
      rz = rxryrz[2]
      point_1 = p[x, y, z, rx, ry, rz]

      x = pointintersect[0] + l2delxunit * rod
      y = pointintersect[1] + l2delyunit * rod
      point_2 = p[x, y, z, rx, ry, rz]

      # now we have the unit vector. extend the weld distance from the intersection
      x = pointintersect[0] + l1delxunit * wd3
      y = pointintersect[1] + l1delyunit * wd3
      # convert the headings to rxryrz and insert those values into the relevant points
      rxryrz = convert_heading_to_axang_ccw(heading1)
      rx = rxryrz[0]
      ry = rxryrz[1]
      rz = rxryrz[2]
      point_5 = p[x, y, z, rx, ry, rz]

      x = pointintersect[0] + l1delxunit * rod
      y = pointintersect[1] + l1delyunit * rod
      point_4 = p[x, y, z, rx, ry, rz]

      #FIND POINT 3
      # by calling analyze_touchpoints()
      atret = analyze_touchpoints(point_2, point_1, point_4, point_5, pointintersect)
      point_3 = atret[5]
      #point 3 will not have the correct rxryrz though because now the gun needs to be face up.
      rxryrz = convert_heading_to_axang_ccw(heading2)
      rx = rxryrz[0]
      ry = rxryrz[1]
      rz = rxryrz[2]
      point_3 = p[point_3[0], point_3[1], point_3[2], rx, ry, rz]

      struct2 = struct(point1=point1, point2=point2, point4=point4, point5=point5, point_1=point_1, point_2=point_2, point_3=point_3, point_4=point_4, point_5=point_5)
      return struct2
  end

  # given a struct from analyze_touchpoints_only(), calculate the points
  # for right, for extended
  def calculate_DOtA_points_right_extended(struct1, listleans, chamferover, chamferup, tcp_pose_top):
      # get the stuff from the struct
      pointintersect = struct1[0]
      heading1 = struct1[1]
      heading2 = struct1[2]
      heading3 = struct1[3]
      l1delxunit = struct1[4]
      l1delyunit = struct1[5]
      l2delxunit = struct1[6]
      l2delyunit = struct1[7]

      # FIND THE POINTS ON THE LINES OF THE FIRST TURN PATH
      # find locations 8 inches away from  intersect point
      # CONST
      # welddistance1 = 8 # vertical weld distance
      welddistance2 = 6 # first path second leg
      welddistance3 = 8 # second path second leg

      # inches
      # wd1 = welddistance1 * 25.4 / 1000
      wd2 = welddistance2 * 25.4 / 1000
      wd3 = welddistance3 * 25.4 / 1000
      zup = chamferup * 25.4 / 1000
      chamferovermm =  chamferover * 25.4 / 1000

      # weld distance is the distance that it will weld. this will make it start at the z height that the user specified
      wd1 = tcp_pose_top[2] - pointintersect[2] - zup

      x = pointintersect[0] + l1delxunit * chamferovermm
      y = pointintersect[1] + l1delyunit * chamferovermm
      z = pointintersect[2] + zup

      #apply actual rxryrz to points
      # convert the headings to rxryrz and insert those values into the relevant points
      rxryrz = convert_heading_to_axang_preheatdown(heading1)
      rx = rxryrz[0]
      ry = rxryrz[1]
      rz = rxryrz[2]

      point1 = p[x + wd1*listleans[0], y + wd1*listleans[1], z + wd1, rx, ry, rz] # add in the listleans factor to follow the face of the box as we move up
      point2 = p[x, y, z, rx, ry, rz]

      # convert the headings to rxryrz and insert those values into the relevant points
      rxryrz = convert_heading_to_axang_ccw(heading1)
      rx = rxryrz[0]
      ry = rxryrz[1]
      rz = rxryrz[2]

      point4 = p[x, y, z, rx, ry, rz]
      x = x + l1delxunit * wd2
      y = y + l1delyunit * wd2
      point5 = p[x, y, z, rx, ry, rz]

      # FIND THE POINTS ON THE LINES OF THE SECOND AROUND PATH
      roundoverdistance = 0.05
      rod = roundoverdistance * 25.4 / 1000

      # now we have the unit vector. extend the weld distance from the intersection
      x = pointintersect[0] + l1delxunit * chamferovermm
      y = pointintersect[1] + l1delyunit * chamferovermm
      # convert the headings to rxryrz and insert those values into the relevant points
      rxryrz = convert_heading_to_axang(heading1)
      rx = rxryrz[0]
      ry = rxryrz[1]
      rz = rxryrz[2]
      point_1 = p[x, y, z, rx, ry, rz]

      x = pointintersect[0] + l1delxunit * rod
      y = pointintersect[1] + l1delyunit * rod
      point_2 = p[x, y, z, rx, ry, rz]

      # convert the headings to rxryrz and insert those values into the relevant points
      rxryrz = convert_heading_to_axang(heading3)
      rx = rxryrz[0]
      ry = rxryrz[1]
      rz = rxryrz[2]

      x = pointintersect[0] + l2delxunit * rod
      y = pointintersect[1] + l2delyunit * rod
      point_4 = p[x, y, z, rx, ry, rz]

      # now we have the unit vector. extend the weld distance from the intersection
      x = pointintersect[0] + l2delxunit * wd3
      y = pointintersect[1] + l2delyunit * wd3
      point_5 = p[x, y, z, rx, ry, rz]

      #FIND POINT 3
      # by calling analyze_touchpoints()
      atret = analyze_touchpoints(point_2, point_1, point_4, point_5, pointintersect)
      atret5 = atret[5]
      point_3 = p[atret5[0], atret5[1], z, atret5[3], atret5[4], atret5[5]]


      struct2 = struct(point1=point1, point2=point2, point4=point4, point5=point5, point_1=point_1, point_2=point_2, point_3=point_3, point_4=point_4, point_5=point_5)
      return struct2
  end

  # given a struct from analyze_touchpoints_only(), calculate the points
  # for left, for extended
  def calculate_DOtA_points_left_extended(struct1, listleans, chamferover, chamferup, tcp_pose_top):
      # get the stuff from the struct
      pointintersect = struct1[0]
      heading1 = struct1[1]
      heading2 = struct1[2]
      heading3 = struct1[3]
      l1delxunit = struct1[4]
      l1delyunit = struct1[5]
      l2delxunit = struct1[6]
      l2delyunit = struct1[7]

      # FIND THE POINTS ON THE LINES OF THE FIRST TURN PATH
      # find locations 8 inches away from  intersect point
      # CONST
      # welddistance1 = 8 # vertical weld distance
      welddistance2 = 6 # first path second leg
      welddistance3 = 8 # second path second leg

      # inches
      # wd1 = welddistance1 * 25.4 / 1000
      wd2 = welddistance2 * 25.4 / 1000
      wd3 = welddistance3 * 25.4 / 1000
      zup = chamferup * 25.4 / 1000
      chamferovermm =  chamferover * 25.4 / 1000

      # weld distance is the distance that it will weld. this will make it start at the z height that the user specified
      wd1 = tcp_pose_top[2] - pointintersect[2] - zup

      x = pointintersect[0] + l2delxunit * chamferovermm
      y = pointintersect[1] + l2delyunit * chamferovermm
      z = pointintersect[2] + zup

      #apply actual rxryrz to points
      # convert the headings to rxryrz and insert those values into the relevant points
      rxryrz = convert_heading_to_axang_preheatdown(heading3)
      rx = rxryrz[0]
      ry = rxryrz[1]
      rz = rxryrz[2]

      point1 = p[x + wd1*listleans[0], y + wd1*listleans[1], z + wd1, rx, ry, rz]
      point2 = p[x, y, z, rx, ry, rz]

      # convert the headings to rxryrz and insert those values into the relevant points
      rxryrz = convert_heading_to_axang(heading3)
      rx = rxryrz[0]
      ry = rxryrz[1]
      rz = rxryrz[2]

      point4 = p[x, y, z, rx, ry, rz]
      x = x + l2delxunit * wd2
      y = y + l2delyunit * wd2
      point5 = p[x, y, z, rx, ry, rz]

      # FIND THE POINTS ON THE LINES OF THE SECOND AROUND PATH
      roundoverdistance = 0.05
      rod = roundoverdistance * 25.4 / 1000

      # now we have the unit vector. extend the weld distance from the intersection
      x = pointintersect[0] + l2delxunit * chamferovermm
      y = pointintersect[1] + l2delyunit * chamferovermm
      # convert the headings to rxryrz and insert those values into the relevant points
      rxryrz = convert_heading_to_axang_ccw(heading3)
      rx = rxryrz[0]
      ry = rxryrz[1]
      rz = rxryrz[2]
      point_1 = p[x, y, z, rx, ry, rz]

      x = pointintersect[0] + l2delxunit * rod
      y = pointintersect[1] + l2delyunit * rod
      point_2 = p[x, y, z, rx, ry, rz]

      # convert the headings to rxryrz and insert those values into the relevant points
      rxryrz = convert_heading_to_axang_ccw(heading1)
      rx = rxryrz[0]
      ry = rxryrz[1]
      rz = rxryrz[2]

      x = pointintersect[0] + l1delxunit * rod
      y = pointintersect[1] + l1delyunit * rod
      point_4 = p[x, y, z, rx, ry, rz]

      # now we have the unit vector. extend the weld distance from the intersection
      x = pointintersect[0] + l1delxunit * wd3
      y = pointintersect[1] + l1delyunit * wd3
      point_5 = p[x, y, z, rx, ry, rz]

      #FIND POINT 3
      # by calling analyze_touchpoints()
      atret = analyze_touchpoints(point_2, point_1, point_4, point_5, pointintersect)
      point_3 = atret[5]
      #point 3 will not have the correct rxryrz though because now the gun needs to be face up
      rxryrz = convert_heading_to_axang_ccw(heading2)
      rx = rxryrz[0]
      ry = rxryrz[1]
      rz = rxryrz[2]
      point_3 = p[point_3[0], point_3[1], z, rx, ry, rz]

      struct2 = struct(point1=point1, point2=point2, point4=point4, point5=point5, point_1=point_1, point_2=point_2, point_3=point_3, point_4=point_4, point_5=point_5)
      return struct2
  end

  # this function analyzes the vertical points
  # calculates the slope of the edge in question
  # specifically, for each inch up in the z direction, what is the change in x and change in y direction
  # returns a list of [nx, ny]
  def analyze_vertical_touchpoints(p11, p12, p13, p21, p22, p23, p3):
      # first, find the equations of the planes from the 6 points
      plane1 = findplane(p11, p12, p13)
      plane2 = findplane(p21, p22, p23)
      # Find the Direction Vector of the Line: The direction vector d of the line of intersection can be found by taking the cross product of the normal vectors of each plane (a, b, and c)
      nx = plane1[1]*plane2[2] - plane1[2]*plane2[1]
      ny = plane1[2]*plane2[0] - plane1[0]*plane2[2]
      nz = plane1[0]*plane2[1] - plane1[1]*plane2[0]
      # normalize the vector so the z length is 1
      multiplier = 1 / nz
      nx = nx * multiplier
      ny = ny * multiplier
      nz = nz * multiplier # should become equal to 1
      ret = [nx, ny]
      return ret
  end

  # given 3 points, this finds the plane and its equation
  # rereturns ax + by + cz + d = 0 in a list of [a, b, c, d]
  def findplane(p11, p12, p13):
      # extract coordinates
      x1 = p11[0]
      y1 = p11[1]
      z1 = p11[2]
      x2 = p12[0]
      y2 = p12[1]
      z2 = p12[2]
      x3 = p13[0]
      y3 = p13[1]
      z3 = p13[2]
      # create vectors from the points
      v1x = x2-x1
      v1y = y2-y1
      v1z = z2-z1
      v2x = x3-x1
      v2y = y3-y1
      v2z = z3-z1
      #calculate the normal vector using the cross product
      nx = v1y*v2z - v1z*v2y # i component
      ny = v1z*v2x - v1x*v2z # j component
      nz = v1x*v2y - v1y*v2x # k component
      # calculate d in the plane equation
      d = -1 * (nx*x1 + ny*y1 + nz*z1)
      ret = [nx, ny, nz, d]
      return ret
  end

  # given a heading, (ccw from +x axis), find the mx+b slope
  # fails if exactly vertical
  def get_slope_from_heading(heading):
      return tan(heading)
  end



  # this function finds the points (and rxryrz) of the 2 points (start and end) of vertical weld section
  def find_vertical_points(pointintersect, l1delxunit, l1delyunit, l2delxunit, l2delyunit, offset, wd, heading1, heading3):

    # find right side stuff
    # find the point in 3d space that is .375 up and .375 over
    x = pointintersect[0] + l1delxunit * offset
    y = pointintersect[1] + l1delyunit * offset
    z = pointintersect[2] + offset
    # find rxryrz
    rxryrz = convert_heading_to_axang_preheatup(heading1)
    rx = rxryrz[0]
    ry = rxryrz[1]
    rz = rxryrz[2]
    path2r1 = p[x, y, z, rx, ry, rz]
    path2r2 = p[x, y, z + wd, rx, ry, rz]

    # find left side
    # find the point in 3d space that is .375 up and .375 over
    x = pointintersect[0] + l2delxunit * offset
    y = pointintersect[1] + l2delyunit * offset
    z = pointintersect[2] + offset
    # find rxryrz
    rxryrz = convert_heading_to_axang_preheatup(heading3)
    rx = rxryrz[0]
    ry = rxryrz[1]
    rz = rxryrz[2]
    path2l1 = p[x, y, z, rx, ry, rz]
    path2l2 = p[x, y, z + wd, rx, ry, rz]

    ret = struct(path2r1=path2r1, path2r2=path2r2, path2l1=path2l1, path2l2=path2l2)
    return ret
  end

  # this function converts a unit vector to its heading angle ccw from x+ axis
  # takes uvx and uvy
  # returns heading in radians
  def convert_uv_to_heading(uvx, uvy):
    baseang = atan(uvy/uvx)
    if uvx < 0:
      ang = baseang + pi
    elif uvy < 0:
      ang = baseang + pi * 2
    else:
      ang = baseang
    end
    return ang
  end

  # this function finds the equation of a line, perpendicular to a given line, and going through a given point
  # takes 3 arguments: m (the original line's slope), x (point's x coord), y (point's y coord). the b of the original line is not needed
  # returns a list of [m,b] (the slope and intercept of the new line)
  def find_perpendicular_line(origm, x, y):
    m = (1/origm) * -1
    b = y - m*x
    ret = [m, b]
    return ret
  end

  # this function finds the intersection point between two lines in the xy plane
  # takes 4 arguments: m1, b1, m2, b2
  # returns a list of [x,y] (the point of intersection)
  def find_intersection(m1, b1, m2, b2):
    # m1x+b1 = m2x+b2
    # m1x - m2x = b2 - b1
    # x = (b2-b1) / (m1-m2)
    x = (b2-b1) / (m1-m2)
    y = m1 * x + b1
    ret = [x, y]
    return ret
  end

  # this function finds the distance between 2 points in 3d space
  # it takes 6 arguments: x1, y1, z1, x2, y2, z2
  # it returns a distance
  def distance_between(x1, y1, z1, x2, y2, z2):
    distsquared = (x2-x1)*(x2-x1)+(y2-y1)*(y2-y1)+(z2-z1)*(z2-z1)
    dist = sqrt(distsquared)
    return dist
  end

  # this function takes a point, a unit vector, and a distance, and adds the distance to the point in the direction of the unit vector (3d space)
  # it returns a point as a list of coordinates
  def add_vectordistance_to_point(xi, yi, zi, uvx, uvy, uvz, delta):
    xf = xi + uvx * delta
    yf = yi + uvy * delta
    zf = zi + uvz * delta
    ret = [xf, yf, zf]
    return ret
  end

  # this function converts a heading (ccw radians from the positive x axis) into rxryrz to be put into a point p[]
  # this will point the gun in this heading with the bottom side of the gun facing up.
  # the values used in this program were calculated by doing rotation matrix math in the file on WI-CALVINB10 C. Documents. Theory for converting rotations into axis angle representations
  def convert_heading_to_axang(heading):
   axisxraw = -1 * sin(heading)
   axisyraw = cos(heading) + 1
   axiszraw = sin(heading)

   magnitude = sqrt(axisxraw*axisxraw + axisyraw*axisyraw + axiszraw*axiszraw)

   axisxunit = axisxraw / magnitude
   axisyunit = axisyraw / magnitude
   axiszunit = axiszraw / magnitude

   angle = acos( (cos(heading) - 1) / 2 )

   rxout = axisxunit * angle
   ryout = axisyunit * angle
   rzout = axiszunit * angle

   return [rxout, ryout, rzout]
  end

  # this function converts a heading (ccw radians from the positive x axis) into rxryrz to be put into a point p[]
  # this will point the gun in this heading with the preheat side of the gun tip facing up. Used for welding in a vertical path.
  # the values used in this program were calculated by doing rotation matrix math in the file on WI-CALVINB10 C. Documents. Theory for converting rotations into axis angle representations
  def convert_heading_to_axang_preheatup(heading):
   axisxraw = -sin(heading) + 1
   axisyraw = cos(heading)
   axiszraw = cos(heading)

   magnitude = sqrt(axisxraw*axisxraw + axisyraw*axisyraw + axiszraw*axiszraw)

   axisxunit = axisxraw / magnitude
   axisyunit = axisyraw / magnitude
   axiszunit = axiszraw / magnitude

   angle = acos( (-sin(heading) - 1) / 2 )

   rxout = axisxunit * angle
   ryout = axisyunit * angle
   rzout = axiszunit * angle

   return [rxout, ryout, rzout]
  end

  # this function converts a heading (ccw radians from the positive x axis) into rxryrz to be put into a point p[]
  # this will point the gun in this heading with the preheat side of the gun tip facing down. Used for welding in a vertical path downwards.
  # the values used in this program were calculated by doing rotation matrix math in the file on WI-CALVINB10 C. Documents. Theory for converting rotations into axis angle representations
  def convert_heading_to_axang_preheatdown(heading):
   axisxraw = -sin(heading) - 1
   axisyraw = cos(heading)
   axiszraw = -cos(heading)

   magnitude = sqrt(axisxraw*axisxraw + axisyraw*axisyraw + axiszraw*axiszraw)

   axisxunit = axisxraw / magnitude
   axisyunit = axisyraw / magnitude
   axiszunit = axiszraw / magnitude

   angle = acos( (sin(heading) - 1) / 2 )

   rxout = axisxunit * angle
   ryout = axisyunit * angle
   rzout = axiszunit * angle

   return [rxout, ryout, rzout]
  end

  # this function converts a heading (ccw radians from the positive x axis) into rxryrz to be put into a point p[]
  # this will point the gun in this heading with the preheat side of the gun tip facing right. Used for welding counterclockwise around the box.
  # the values used in this program were calculated by doing rotation matrix math in the file on WI-CALVINB10 C. Documents. Theory for converting rotations into axis angle representations
  def convert_heading_to_axang_ccw(heading):
   axisxraw = -sin(heading)
   axisyraw = cos(heading) - 1
   axiszraw = -sin(heading)

   magnitude = sqrt(axisxraw*axisxraw + axisyraw*axisyraw + axiszraw*axiszraw)

   axisxunit = axisxraw / magnitude
   axisyunit = axisyraw / magnitude
   axiszunit = axiszraw / magnitude

   angle = acos( (-cos(heading) - 1) / 2 )

   rxout = axisxunit * angle
   ryout = axisyunit * angle
   rzout = axiszunit * angle

   return [rxout, ryout, rzout]
  end

  # this function is for getting the points along the path of the corner homing 45
  # point0 is the point where they touched
  def get_corner_homing_45_pathpoints(point0, pointtop = p[0,0,0,0,0,0]):
    p0x = point0[0]
    p0y = point0[1]
    p0z = point0[2]
    p0rx = point0[3]
    p0ry = point0[4]
    p0rz = point0[5]

    #constants
    #distances of how far away from point the touchpoints are
    d0 = 0.10 # how far from the box to retreat and approach
    d1 = 0.06 # first distance from init point
    d2 = 0.15 # second distance from init point
    d3 = 0.125 #vertical distance from first point
    sqrt2 = 0.707106781 # 1/sqrt(2) , the inverse of the sqrt(2)

    ph1 = p[p0x + d0, p0y, p0z + d1, p0rx, p0ry, p0rz] #approach point for turn

    ph2 = p[p0x+d0-d0*0.5-sqrt2*d1, p0y+d0*0.5+sqrt2*d1, p0z+d1, 1.446, -0.8, -0.733]
    ph3 = p[p0x+d0-d0*0.5-sqrt2*d2, p0y+d0*0.5+sqrt2*d2, p0z+d1, 1.446, -0.8, -0.733]
    ph4 = p[p0x+d0-d0*0.5-sqrt2*d1, p0y-d0*0.5-sqrt2*d1, p0z+d1, 0.626, -1.993, -1.813]
    ph5 = p[p0x+d0-d0*0.5-sqrt2*d2, p0y-d0*0.5-sqrt2*d2, p0z+d1, 0.626, -1.993, -1.813]

